LIN {X 0,Y 575.215,Z 1088.939,A -85,B 0,C 180,E1 20584.216,E2 20584.216} C_VEL
LIN {X 0,Y 578.053,Z 1069.285,A -85,B 0,C 180,E1 20581.709,E2 20581.709} C_VEL
LIN {X 0,Y 580.453,Z 1053.893,A -85,B 0,C 180,E1 20579.973,E2 20579.973} C_VEL
LIN {X 0,Y 583.494,Z 1035.186,A -85,B 0,C 180,E1 20578.086,E2 20578.086} C_VEL
LIN {X 0,Y 586.743,Z 1014.887,A -85,B 0,C 180,E1 20576.311,E2 20576.311} C_VEL
LIN {X 0,Y 589.518,Z 997.438,A -85,B 0,C 180,E1 20574.962,E2 20574.962} C_VEL
LIN {X 0,Y 592.71,Z 977.137,A -85,B 0,C 180,E1 20573.573,E2 20573.573} C_VEL
LIN {X 0,Y 595.995,Z 954.418,A -85,B 0,C 180,E1 20572.241,E2 20572.241} C_VEL
LIN {X 0,Y 598.554,Z 935.209,A -85,B 0,C 180,E1 20571.273,E2 20571.273} C_VEL
LIN {X 0,Y 600.798,Z 916.678,A -85,B 0,C 180,E1 20570.463,E2 20570.463} C_VEL
LIN {X 0,Y 603.05,Z 895.538,A -85,B 0,C 180,E1 20569.681,E2 20569.681} C_VEL
LIN {X 0,Y 605.325,Z 869.865,A -85,B 0,C 180,E1 20568.921,E2 20568.921} C_VEL
LIN {X 0,Y 606.783,Z 848.524,A -85,B 0,C 180,E1 20568.434,E2 20568.434} C_VEL
LIN {X 0,Y 607.837,Z 827.107,A -85,B 0,C 180,E1 20568.062,E2 20568.062} C_VEL
LIN {X 0,Y 613.605,Z 599.561,A -85,B 0,C 180,E1 20564.976,E2 20564.976} C_VEL
LIN {X 0,Y 617.781,Z 441.673,A -85,B 0,C 180,E1 20562.787,E2 20562.787} C_VEL
LIN {X 0,Y 611.446,Z 410.233,A -85,B 0,C 180,E1 20561.538,E2 20561.538} C_VEL
LIN {X 0,Y 597.897,Z 389.86,A -85,B 0,C 180,E1 20559.519,E2 20559.519} C_VEL
LIN {X 0,Y 590.526,Z 374.156,A -85,B 0,C 180,E1 20557.07,E2 20557.07} C_VEL
LIN {X 0,Y 583.564,Z 360.458,A -85,B 0,C 180,E1 20554.671,E2 20554.671} C_VEL
LIN {X 0,Y 579.173,Z 351.956,A -85,B 0,C 180,E1 20553.062,E2 20553.062} C_VEL
LIN {X 0,Y 576.456,Z 347.036,A -85,B 0,C 180,E1 20552.058,E2 20552.058} C_VEL
LIN {X 0,Y 574.452,Z 343.015,A -85,B 0,C 180,E1 20551.245,E2 20551.245} C_VEL
LIN {X 0,Y 572.351,Z 339.399,A -85,B 0,C 180,E1 20550.44,E2 20550.44} C_VEL
LIN {X 0,Y 571.332,Z 337.612,A -85,B 0,C 180,E1 20550.035,E2 20550.035} C_VEL
LIN {X 0,Y 569.492,Z 333.982,A -85,B 0,C 180,E1 20549.216,E2 20549.216} C_VEL
LIN {X 0,Y 569.352,Z 333.336,A -85,B 0,C 180,E1 20548.879,E2 20548.879} C_VEL
LIN {X 0,Y 569.379,Z 333.282,A -85,B 0,C 180,E1 20545.595,E2 20545.595} C_VEL
LIN {X 0,Y 569.349,Z 333.278,A -85,B 0,C 180,E1 20542.293,E2 20542.293} C_VEL
LIN {X 0,Y 569.372,Z 333.252,A -85,B 0,C 180,E1 20539.065,E2 20539.065} C_VEL
LIN {X 0,Y 569.379,Z 333.308,A -85,B 0,C 180,E1 20535.691,E2 20535.691} C_VEL
LIN {X 0,Y 569.354,Z 333.245,A -85,B 0,C 180,E1 20532.372,E2 20532.372} C_VEL
LIN {X 0,Y 569.369,Z 333.302,A -85,B 0,C 180,E1 20529.094,E2 20529.094} C_VEL
LIN {X 0,Y 569.369,Z 333.245,A -85,B 0,C 180,E1 20525.745,E2 20525.745} C_VEL
LIN {X 0,Y 569.374,Z 333.291,A -85,B 0,C 180,E1 20522.416,E2 20522.416} C_VEL
LIN {X 0,Y 569.352,Z 333.257,A -85,B 0,C 180,E1 20519.094,E2 20519.094} C_VEL
LIN {X 0,Y 569.373,Z 333.284,A -85,B 0,C 180,E1 20515.871,E2 20515.871} C_VEL
LIN {X 0,Y 569.359,Z 333.264,A -85,B 0,C 180,E1 20512.533,E2 20512.533} C_VEL
LIN {X 0,Y 569.349,Z 333.267,A -85,B 0,C 180,E1 20509.169,E2 20509.169} C_VEL
LIN {X 0,Y 569.382,Z 333.284,A -85,B 0,C 180,E1 20505.871,E2 20505.871} C_VEL
LIN {X 0,Y 569.332,Z 333.255,A -85,B 0,C 180,E1 20502.629,E2 20502.629} C_VEL
LIN {X 0,Y 569.371,Z 333.311,A -85,B 0,C 180,E1 20499.33,E2 20499.33} C_VEL
LIN {X 0,Y 569.337,Z 333.257,A -85,B 0,C 180,E1 20496.175,E2 20496.175} C_VEL
LIN {X 0,Y 569.327,Z 333.282,A -85,B 0,C 180,E1 20492.83,E2 20492.83} C_VEL
LIN {X 0,Y 569.39,Z 333.734,A -85,B 0,C 180,E1 20492.411,E2 20492.411} C_VEL
LIN {X 0,Y 570.987,Z 337.158,A -85,B 0,C 180,E1 20491.669,E2 20491.669} C_VEL
LIN {X 0,Y 572.36,Z 339.239,A -85,B 0,C 180,E1 20491.173,E2 20491.173} C_VEL
LIN {X 0,Y 574.43,Z 343,A -85,B 0,C 180,E1 20490.373,E2 20490.373} C_VEL
LIN {X 0,Y 577.912,Z 349.337,A -85,B 0,C 180,E1 20489.078,E2 20489.078} C_VEL
LIN {X 0,Y 582.608,Z 357.641,A -85,B 0,C 180,E1 20487.508,E2 20487.508} C_VEL
LIN {X 0,Y 592.791,Z 370.97,A -85,B 0,C 180,E1 20485.827,E2 20485.827} C_VEL
LIN {X 0,Y 602.215,Z 383.402,A -85,B 0,C 180,E1 20484.382,E2 20484.382} C_VEL
LIN {X 0,Y 615.574,Z 402.306,A -85,B 0,C 180,E1 20482.459,E2 20482.459} C_VEL
LIN {X 0,Y 622.733,Z 413.094,A -85,B 0,C 180,E1 20481.481,E2 20481.481} C_VEL
LIN {X 0,Y 616.942,Z 613.718,A -85,B 0,C 180,E1 20478.606,E2 20478.606} C_VEL
LIN {X 0,Y 611.425,Z 825.012,A -85,B 0,C 180,E1 20475.663,E2 20475.663} C_VEL
LIN {X 0,Y 610.25,Z 847.871,A -85,B 0,C 180,E1 20475.265,E2 20475.265} C_VEL
LIN {X 0,Y 608.433,Z 874.998,A -85,B 0,C 180,E1 20474.636,E2 20474.636} C_VEL
LIN {X 0,Y 606.238,Z 899.951,A -85,B 0,C 180,E1 20473.882,E2 20473.882} C_VEL
LIN {X 0,Y 604.145,Z 921.03,A -85,B 0,C 180,E1 20473.12,E2 20473.12} C_VEL
LIN {X 0,Y 601.971,Z 941.046,A -85,B 0,C 180,E1 20472.276,E2 20472.276} C_VEL
LIN {X 0,Y 599.598,Z 960.799,A -85,B 0,C 180,E1 20471.327,E2 20471.327} C_VEL
LIN {X 0,Y 596.742,Z 983.005,A -85,B 0,C 180,E1 20470.109,E2 20470.109} C_VEL
LIN {X 0,Y 593.087,Z 1007.09,A -85,B 0,C 180,E1 20468.531,E2 20468.531} C_VEL
LIN {X 0,Y 590.071,Z 1026.218,A -85,B 0,C 180,E1 20467.102,E2 20467.102} C_VEL
LIN {X 0,Y 587.305,Z 1043.431,A -85,B 0,C 180,E1 20465.669,E2 20465.669} C_VEL
LIN {X 0,Y 584.512,Z 1060.71,A -85,B 0,C 180,E1 20464.071,E2 20464.071} C_VEL
LIN {X 0,Y 581.227,Z 1081.272,A -85,B 0,C 180,E1 20461.937,E2 20461.937} C_VEL
LIN {X 0,Y 578.488,Z 1098.828,A -85,B 0,C 180,E1 20459.854,E2 20459.854} C_VEL
LIN {X 0,Y 576.301,Z 1113.378,A -85,B 0,C 180,E1 20457.933,E2 20457.933} C_VEL
LIN {X 0,Y 574.059,Z 1129.58,A -85,B 0,C 180,E1 20455.544,E2 20455.544} C_VEL
LIN {X 0,Y 572.164,Z 1144.275,A -85,B 0,C 180,E1 20453.044,E2 20453.044} C_VEL
LIN {X 0,Y 570.861,Z 1155.779,A -85,B 0,C 180,E1 20450.827,E2 20450.827} C_VEL
LIN {X 0,Y 569.844,Z 1166.361,A -85,B 0,C 180,E1 20448.517,E2 20448.517} C_VEL
LIN {X 0,Y 568.941,Z 1177.381,A -85,B 0,C 180,E1 20445.702,E2 20445.702} C_VEL
LIN {X 0,Y 568.479,Z 1185.17,A -85,B 0,C 180,E1 20443.321,E2 20443.321} C_VEL
LIN {X 0,Y 568.159,Z 1191.597,A -85,B 0,C 180,E1 20440.956,E2 20440.956} C_VEL
LIN {X 0,Y 568.007,Z 1197.191,A -85,B 0,C 180,E1 20438.381,E2 20438.381} C_VEL
LIN {X 0,Y 567.933,Z 1201.538,A -85,B 0,C 180,E1 20435.556,E2 20435.556} C_VEL
LIN {X 0,Y 567.917,Z 1203.848,A -85,B 0,C 180,E1 20433.128,E2 20433.128} C_VEL
LIN {X 0,Y 567.906,Z 1204.804,A -85,B 0,C 180,E1 20430.908,E2 20430.908} C_VEL
LIN {X 0,Y 567.916,Z 1204.736,A -85,B 0,C 180,E1 20428.789,E2 20428.789} C_VEL
LIN {X 0,Y 567.912,Z 1203.507,A -85,B 0,C 180,E1 20426.366,E2 20426.366} C_VEL
LIN {X 0,Y 567.948,Z 1200.335,A -85,B 0,C 180,E1 20423.53,E2 20423.53} C_VEL
LIN {X 0,Y 568.029,Z 1196.126,A -85,B 0,C 180,E1 20421.089,E2 20421.089} C_VEL
LIN {X 0,Y 568.191,Z 1190.833,A -85,B 0,C 180,E1 20418.736,E2 20418.736} C_VEL
LIN {X 0,Y 568.577,Z 1183.47,A -85,B 0,C 180,E1 20416.106,E2 20416.106} C_VEL
LIN {X 0,Y 569.205,Z 1173.918,A -85,B 0,C 180,E1 20413.361,E2 20413.361} C_VEL
LIN {X 0,Y 570.006,Z 1164.527,A -85,B 0,C 180,E1 20411.063,E2 20411.063} C_VEL
LIN {X 0,Y 571.044,Z 1154.238,A -85,B 0,C 180,E1 20408.857,E2 20408.857} C_VEL
LIN {X 0,Y 572.692,Z 1140.174,A -85,B 0,C 180,E1 20406.215,E2 20406.215} C_VEL
LIN {X 0,Y 574.534,Z 1125.776,A -85,B 0,C 180,E1 20403.877,E2 20403.877} C_VEL
LIN {X 0,Y 576.538,Z 1111.833,A -85,B 0,C 180,E1 20401.854,E2 20401.854} C_VEL
LIN {X 0,Y 579.024,Z 1095.329,A -85,B 0,C 180,E1 20399.704,E2 20399.704} C_VEL
LIN {X 0,Y 582.167,Z 1075.37,A -85,B 0,C 180,E1 20397.428,E2 20397.428} C_VEL
LIN {X 0,Y 584.784,Z 1059.04,A -85,B 0,C 180,E1 20395.769,E2 20395.769} C_VEL
LIN {X 0,Y 587.477,Z 1042.38,A -85,B 0,C 180,E1 20394.24,E2 20394.24} C_VEL
LIN {X 0,Y 590.375,Z 1024.362,A -85,B 0,C 180,E1 20392.752,E2 20392.752} C_VEL
LIN {X 0,Y 594.049,Z 1001.028,A -85,B 0,C 180,E1 20391.044,E2 20391.044} C_VEL
LIN {X 0,Y 597.088,Z 980.227,A -85,B 0,C 180,E1 20389.73,E2 20389.73} C_VEL
LIN {X 0,Y 599.74,Z 959.604,A -85,B 0,C 180,E1 20388.612,E2 20388.612} C_VEL
LIN {X 0,Y 602.123,Z 939.747,A -85,B 0,C 180,E1 20387.666,E2 20387.666} C_VEL
LIN {X 0,Y 604.431,Z 918.348,A -85,B 0,C 180,E1 20386.775,E2 20386.775} C_VEL
LIN {X 0,Y 607.062,Z 891.208,A -85,B 0,C 180,E1 20385.832,E2 20385.832} C_VEL
LIN {X 0,Y 609.036,Z 866.174,A -85,B 0,C 180,E1 20385.144,E2 20385.144} C_VEL
LIN {X 0,Y 610.419,Z 844.794,A -85,B 0,C 180,E1 20384.674,E2 20384.674} C_VEL
LIN {X 0,Y 611.52,Z 822.48,A -85,B 0,C 180,E1 20384.299,E2 20384.299} C_VEL
LIN {X 0,Y 617.232,Z 602.035,A -85,B 0,C 180,E1 20381.232,E2 20381.232} C_VEL
LIN {X 0,Y 622.721,Z 412.863,A -85,B 0,C 180,E1 20378.514,E2 20378.514} C_VEL
LIN {X 0,Y 607.623,Z 390.884,A -85,B 0,C 180,E1 20376.416,E2 20376.416} C_VEL
LIN {X 0,Y 594.34,Z 372.937,A -85,B 0,C 180,E1 20374.421,E2 20374.421} C_VEL
LIN {X 0,Y 586.055,Z 362.24,A -85,B 0,C 180,E1 20373.091,E2 20373.091} C_VEL
LIN {X 0,Y 582.119,Z 357.051,A -85,B 0,C 180,E1 20372.406,E2 20372.406} C_VEL
LIN {X 0,Y 579.52,Z 352.35,A -85,B 0,C 180,E1 20371.52,E2 20371.52} C_VEL
LIN {X 0,Y 576.62,Z 347.132,A -85,B 0,C 180,E1 20370.479,E2 20370.479} C_VEL
LIN {X 0,Y 574.387,Z 342.955,A -85,B 0,C 180,E1 20369.629,E2 20369.629} C_VEL
LIN {X 0,Y 572.332,Z 339.159,A -85,B 0,C 180,E1 20368.828,E2 20368.828} C_VEL
LIN {X 0,Y 569.532,Z 334.345,A -85,B 0,C 180,E1 20367.726,E2 20367.726} C_VEL
LIN {X 0,Y 569.344,Z 333.479,A -85,B 0,C 180,E1 20367.509,E2 20367.509} C_VEL
LIN {X 0,Y 569.38,Z 333.261,A -85,B 0,C 180,E1 20364.374,E2 20364.374} C_VEL
LIN {X 0,Y 569.331,Z 333.303,A -85,B 0,C 180,E1 20361.162,E2 20361.162} C_VEL
LIN {X 0,Y 569.357,Z 333.249,A -85,B 0,C 180,E1 20357.855,E2 20357.855} C_VEL
LIN {X 0,Y 569.367,Z 333.303,A -85,B 0,C 180,E1 20354.619,E2 20354.619} C_VEL
LIN {X 0,Y 569.339,Z 333.255,A -85,B 0,C 180,E1 20351.344,E2 20351.344} C_VEL
LIN {X 0,Y 569.377,Z 333.289,A -85,B 0,C 180,E1 20348.178,E2 20348.178} C_VEL
LIN {X 0,Y 569.344,Z 333.261,A -85,B 0,C 180,E1 20344.937,E2 20344.937} C_VEL
LIN {X 0,Y 569.376,Z 333.281,A -85,B 0,C 180,E1 20341.711,E2 20341.711} C_VEL
LIN {X 0,Y 569.368,Z 333.263,A -85,B 0,C 180,E1 20338.39,E2 20338.39} C_VEL
LIN {X 0,Y 569.359,Z 333.267,A -85,B 0,C 180,E1 20335.063,E2 20335.063} C_VEL
LIN {X 0,Y 569.364,Z 333.27,A -85,B 0,C 180,E1 20331.822,E2 20331.822} C_VEL
LIN {X 0,Y 569.363,Z 333.256,A -85,B 0,C 180,E1 20328.554,E2 20328.554} C_VEL
LIN {X 0,Y 569.381,Z 333.294,A -85,B 0,C 180,E1 20325.144,E2 20325.144} C_VEL
LIN {X 0,Y 569.357,Z 333.249,A -85,B 0,C 180,E1 20321.784,E2 20321.784} C_VEL
LIN {X 0,Y 569.375,Z 333.305,A -85,B 0,C 180,E1 20318.467,E2 20318.467} C_VEL
LIN {X 0,Y 569.35,Z 333.261,A -85,B 0,C 180,E1 20315.182,E2 20315.182} C_VEL
LIN {X 0,Y 569.362,Z 333.258,A -85,B 0,C 180,E1 20311.834,E2 20311.834} C_VEL
LIN {X 0,Y 569.43,Z 333.642,A -85,B 0,C 180,E1 20310.739,E2 20310.739} C_VEL
LIN {X 0,Y 571.05,Z 337.255,A -85,B 0,C 180,E1 20309.948,E2 20309.948} C_VEL
LIN {X 0,Y 572.364,Z 339.417,A -85,B 0,C 180,E1 20309.445,E2 20309.445} C_VEL
LIN {X 0,Y 574.475,Z 343.031,A -85,B 0,C 180,E1 20308.64,E2 20308.64} C_VEL
LIN {X 0,Y 577.257,Z 348.085,A -85,B 0,C 180,E1 20307.581,E2 20307.581} C_VEL
LIN {X 0,Y 584.777,Z 362.651,A -85,B 0,C 180,E1 20304.814,E2 20304.814} C_VEL
LIN {X 0,Y 591.129,Z 375.567,A -85,B 0,C 180,E1 20302.609,E2 20302.609} C_VEL
LIN {X 0,Y 598.317,Z 390.561,A -85,B 0,C 180,E1 20300.297,E2 20300.297} C_VEL
LIN {X 0,Y 611.582,Z 410.455,A -85,B 0,C 180,E1 20298.348,E2 20298.348} C_VEL
LIN {X 0,Y 617.828,Z 442.453,A -85,B 0,C 180,E1 20297.101,E2 20297.101} C_VEL
LIN {X 0,Y 612.398,Z 646.343,A -85,B 0,C 180,E1 20294.298,E2 20294.298} C_VEL
LIN {X 0,Y 611.526,Z 654.049,A -85,B 0,C 180,E1 20294.26,E2 20294.26} C_VEL
LIN {X 0,Y 606.683,Z 674.681,A -85,B 0,C 180,E1 20294.41,E2 20294.41} C_VEL
LIN {X 0,Y 605.99,Z 681.294,A -85,B 0,C 180,E1 20294.372,E2 20294.372} C_VEL
LIN {X 0,Y 601.978,Z 831.027,A -85,B 0,C 180,E1 20292.324,E2 20292.324} C_VEL
LIN {X 0,Y 600.473,Z 857.229,A -85,B 0,C 180,E1 20291.836,E2 20291.836} C_VEL
LIN {X 0,Y 598.478,Z 881.561,A -85,B 0,C 180,E1 20291.203,E2 20291.203} C_VEL
LIN {X 0,Y 596.403,Z 902.748,A -85,B 0,C 180,E1 20290.515,E2 20290.515} C_VEL
LIN {X 0,Y 593.623,Z 927.269,A -85,B 0,C 180,E1 20289.546,E2 20289.546} C_VEL
LIN {X 0,Y 590.628,Z 949.512,A -85,B 0,C 180,E1 20288.473,E2 20288.473} C_VEL
LIN {X 0,Y 587.921,Z 967.877,A -85,B 0,C 180,E1 20287.445,E2 20287.445} C_VEL
LIN {X 0,Y 584.637,Z 988.821,A -85,B 0,C 180,E1 20286.099,E2 20286.099} C_VEL
LIN {X 0,Y 580.995,Z 1010.481,A -85,B 0,C 180,E1 20284.476,E2 20284.476} C_VEL
LIN {X 0,Y 578.043,Z 1027.611,A -85,B 0,C 180,E1 20283.016,E2 20283.016} C_VEL
LIN {X 0,Y 575.112,Z 1044.691,A -85,B 0,C 180,E1 20281.388,E2 20281.388} C_VEL
LIN {X 0,Y 571.696,Z 1064.709,A -85,B 0,C 180,E1 20279.207,E2 20279.207} C_VEL
LIN {X 0,Y 569.31,Z 1079.368,A -85,B 0,C 180,E1 20277.397,E2 20277.397} C_VEL
LIN {X 0,Y 567.05,Z 1094.053,A -85,B 0,C 180,E1 20275.371,E2 20275.371} C_VEL
LIN {X 0,Y 564.814,Z 1110.511,A -85,B 0,C 180,E1 20272.811,E2 20272.811} C_VEL
LIN {X 0,Y 563.394,Z 1122.352,A -85,B 0,C 180,E1 20270.722,E2 20270.722} C_VEL
LIN {X 0,Y 562.109,Z 1134.782,A -85,B 0,C 180,E1 20268.214,E2 20268.214} C_VEL
LIN {X 0,Y 561.215,Z 1144.797,A -85,B 0,C 180,E1 20265.819,E2 20265.819} C_VEL
LIN {X 0,Y 560.651,Z 1152.781,A -85,B 0,C 180,E1 20263.595,E2 20263.595} C_VEL
LIN {X 0,Y 560.226,Z 1160.757,A -85,B 0,C 180,E1 20260.906,E2 20260.906} C_VEL
LIN {X 0,Y 560.04,Z 1166.03,A -85,B 0,C 180,E1 20258.625,E2 20258.625} C_VEL
LIN {X 0,Y 559.956,Z 1169.917,A -85,B 0,C 180,E1 20256.459,E2 20256.459} C_VEL
LIN {X 0,Y 559.914,Z 1172.807,A -85,B 0,C 180,E1 20254.199,E2 20254.199} C_VEL
LIN {X 0,Y 559.902,Z 1174.653,A -85,B 0,C 180,E1 20251.535,E2 20251.535} C_VEL
LIN {X 0,Y 559.897,Z 1174.856,A -85,B 0,C 180,E1 20249.284,E2 20249.284} C_VEL
LIN {X 0,Y 559.906,Z 1173.968,A -85,B 0,C 180,E1 20247.134,E2 20247.134} C_VEL
LIN {X 0,Y 559.916,Z 1171.999,A -85,B 0,C 180,E1 20244.98,E2 20244.98} C_VEL
LIN {X 0,Y 559.979,Z 1168.276,A -85,B 0,C 180,E1 20242.407,E2 20242.407} C_VEL
LIN {X 0,Y 560.122,Z 1163.013,A -85,B 0,C 180,E1 20239.925,E2 20239.925} C_VEL
LIN {X 0,Y 560.401,Z 1157.204,A -85,B 0,C 180,E1 20237.742,E2 20237.742} C_VEL
LIN {X 0,Y 560.842,Z 1149.832,A -85,B 0,C 180,E1 20235.441,E2 20235.441} C_VEL
LIN {X 0,Y 561.64,Z 1139.632,A -85,B 0,C 180,E1 20232.811,E2 20232.811} C_VEL
LIN {X 0,Y 562.562,Z 1130.009,A -85,B 0,C 180,E1 20230.696,E2 20230.696} C_VEL
LIN {X 0,Y 563.78,Z 1119.028,A -85,B 0,C 180,E1 20228.571,E2 20228.571} C_VEL
LIN {X 0,Y 565.678,Z 1103.775,A -85,B 0,C 180,E1 20226.012,E2 20226.012} C_VEL
LIN {X 0,Y 568.094,Z 1087.181,A -85,B 0,C 180,E1 20223.558,E2 20223.558} C_VEL
LIN {X 0,Y 570.85,Z 1069.89,A -85,B 0,C 180,E1 20221.32,E2 20221.32} C_VEL
LIN {X 0,Y 573.487,Z 1054.105,A -85,B 0,C 180,E1 20219.512,E2 20219.512} C_VEL
LIN {X 0,Y 576.522,Z 1036.52,A -85,B 0,C 180,E1 20217.713,E2 20217.713} C_VEL
LIN {X 0,Y 580.176,Z 1015.196,A -85,B 0,C 180,E1 20215.818,E2 20215.818} C_VEL
LIN {X 0,Y 583.119,Z 997.822,A -85,B 0,C 180,E1 20214.459,E2 20214.459} C_VEL
LIN {X 0,Y 586.335,Z 978.32,A -85,B 0,C 180,E1 20213.111,E2 20213.111} C_VEL
LIN {X 0,Y 589.918,Z 954.728,A -85,B 0,C 180,E1 20211.714,E2 20211.714} C_VEL
LIN {X 0,Y 592.557,Z 935.478,A -85,B 0,C 180,E1 20210.745,E2 20210.745} C_VEL
LIN {X 0,Y 594.882,Z 916.705,A -85,B 0,C 180,E1 20209.929,E2 20209.929} C_VEL
LIN {X 0,Y 597.121,Z 896.268,A -85,B 0,C 180,E1 20209.171,E2 20209.171} C_VEL
LIN {X 0,Y 599.501,Z 870.507,A -85,B 0,C 180,E1 20208.402,E2 20208.402} C_VEL
LIN {X 0,Y 601.046,Z 848.667,A -85,B 0,C 180,E1 20207.901,E2 20207.901} C_VEL
LIN {X 0,Y 602.135,Z 827.355,A -85,B 0,C 180,E1 20207.53,E2 20207.53} C_VEL
LIN {X 0,Y 608.258,Z 596.705,A -85,B 0,C 180,E1 20204.381,E2 20204.381} C_VEL
LIN {X 0,Y 612.512,Z 443.576,A -85,B 0,C 180,E1 20202.242,E2 20202.242} C_VEL
LIN {X 0,Y 606.894,Z 415.194,A -85,B 0,C 180,E1 20201.1,E2 20201.1} C_VEL
LIN {X 0,Y 593.37,Z 395.038,A -85,B 0,C 180,E1 20199.067,E2 20199.067} C_VEL
LIN {X 0,Y 589.348,Z 388.963,A -85,B 0,C 180,E1 20198.386,E2 20198.386} C_VEL
LIN {X 0,Y 582.296,Z 374.276,A -85,B 0,C 180,E1 20195.963,E2 20195.963} C_VEL
LIN {X 0,Y 576.415,Z 362.589,A -85,B 0,C 180,E1 20193.837,E2 20193.837} C_VEL
LIN {X 0,Y 571.585,Z 353.4,A -85,B 0,C 180,E1 20192.009,E2 20192.009} C_VEL
LIN {X 0,Y 568.98,Z 348.618,A -85,B 0,C 180,E1 20190.991,E2 20190.991} C_VEL
LIN {X 0,Y 566.206,Z 343.58,A -85,B 0,C 180,E1 20189.868,E2 20189.868} C_VEL
LIN {X 0,Y 563.74,Z 339.019,A -85,B 0,C 180,E1 20188.815,E2 20188.815} C_VEL
LIN {X 0,Y 561.82,Z 335.92,A -85,B 0,C 180,E1 20188.025,E2 20188.025} C_VEL
LIN {X 0,Y 561.468,Z 334.458,A -85,B 0,C 180,E1 20187.656,E2 20187.656} C_VEL
LIN {X 0,Y 561.403,Z 334.243,A -85,B 0,C 180,E1 20184.406,E2 20184.406} C_VEL
LIN {X 0,Y 561.441,Z 334.297,A -85,B 0,C 180,E1 20181.062,E2 20181.062} C_VEL
LIN {X 0,Y 561.433,Z 334.239,A -85,B 0,C 180,E1 20177.674,E2 20177.674} C_VEL
LIN {X 0,Y 561.417,Z 334.27,A -85,B 0,C 180,E1 20174.439,E2 20174.439} C_VEL
LIN {X 0,Y 561.427,Z 334.251,A -85,B 0,C 180,E1 20171.097,E2 20171.097} C_VEL
LIN {X 0,Y 561.434,Z 334.245,A -85,B 0,C 180,E1 20167.779,E2 20167.779} C_VEL
LIN {X 0,Y 561.431,Z 334.271,A -85,B 0,C 180,E1 20164.392,E2 20164.392} C_VEL
LIN {X 0,Y 561.414,Z 334.24,A -85,B 0,C 180,E1 20161.123,E2 20161.123} C_VEL
LIN {X 0,Y 561.434,Z 334.284,A -85,B 0,C 180,E1 20157.857,E2 20157.857} C_VEL
LIN {X 0,Y 561.419,Z 334.236,A -85,B 0,C 180,E1 20154.584,E2 20154.584} C_VEL
LIN {X 0,Y 561.416,Z 334.294,A -85,B 0,C 180,E1 20151.189,E2 20151.189} C_VEL
LIN {X 0,Y 561.434,Z 334.23,A -85,B 0,C 180,E1 20147.869,E2 20147.869} C_VEL
LIN {X 0,Y 561.403,Z 334.299,A -85,B 0,C 180,E1 20144.611,E2 20144.611} C_VEL
LIN {X 0,Y 561.419,Z 334.241,A -85,B 0,C 180,E1 20141.302,E2 20141.302} C_VEL
LIN {X 0,Y 561.409,Z 334.262,A -85,B 0,C 180,E1 20138.146,E2 20138.146} C_VEL
LIN {X 0,Y 561.39,Z 334.28,A -85,B 0,C 180,E1 20134.794,E2 20134.794} C_VEL
LIN {X 0,Y 561.488,Z 334.675,A -85,B 0,C 180,E1 20133.815,E2 20133.815} C_VEL
LIN {X 0,Y 563.184,Z 338.387,A -85,B 0,C 180,E1 20132.967,E2 20132.967} C_VEL
LIN {X 0,Y 564.507,Z 340.35,A -85,B 0,C 180,E1 20132.464,E2 20132.464} C_VEL
LIN {X 0,Y 566.511,Z 343.879,A -85,B 0,C 180,E1 20131.655,E2 20131.655} C_VEL
LIN {X 0,Y 567.71,Z 346.299,A -85,B 0,C 180,E1 20131.145,E2 20131.145} C_VEL
LIN {X 0,Y 570.374,Z 350.886,A -85,B 0,C 180,E1 20130.141,E2 20130.141} C_VEL
LIN {X 0,Y 573.266,Z 356.395,A -85,B 0,C 180,E1 20129.033,E2 20129.033} C_VEL
LIN {X 0,Y 575.118,Z 359.033,A -85,B 0,C 180,E1 20128.562,E2 20128.562} C_VEL
LIN {X 0,Y 585.729,Z 372.597,A -85,B 0,C 180,E1 20126.742,E2 20126.742} C_VEL
LIN {X 0,Y 596.398,Z 386.71,A -85,B 0,C 180,E1 20125.043,E2 20125.043} C_VEL
LIN {X 0,Y 608.942,Z 404.374,A -85,B 0,C 180,E1 20123.178,E2 20123.178} C_VEL
LIN {X 0,Y 617.393,Z 417.147,A -85,B 0,C 180,E1 20121.988,E2 20121.988} C_VEL
LIN {X 0,Y 611.149,Z 620.112,A -85,B 0,C 180,E1 20119.051,E2 20119.051} C_VEL
LIN {X 0,Y 605.333,Z 827.696,A -85,B 0,C 180,E1 20116.126,E2 20116.126} C_VEL
LIN {X 0,Y 603.724,Z 855.846,A -85,B 0,C 180,E1 20115.601,E2 20115.601} C_VEL
LIN {X 0,Y 601.702,Z 881.502,A -85,B 0,C 180,E1 20114.947,E2 20114.947} C_VEL
LIN {X 0,Y 599.75,Z 902.878,A -85,B 0,C 180,E1 20114.276,E2 20114.276} C_VEL
LIN {X 0,Y 597.6,Z 923.472,A -85,B 0,C 180,E1 20113.511,E2 20113.511} C_VEL
LIN {X 0,Y 594.924,Z 946.696,A -85,B 0,C 180,E1 20112.503,E2 20112.503} C_VEL
LIN {X 0,Y 591.532,Z 972.526,A -85,B 0,C 180,E1 20111.176,E2 20111.176} C_VEL
LIN {X 0,Y 588.613,Z 993.178,A -85,B 0,C 180,E1 20109.949,E2 20109.949} C_VEL
LIN {X 0,Y 586.118,Z 1010.033,A -85,B 0,C 180,E1 20108.824,E2 20108.824} C_VEL
LIN {X 0,Y 583.224,Z 1027.551,A -85,B 0,C 180,E1 20107.489,E2 20107.489} C_VEL
LIN {X 0,Y 580.229,Z 1045.255,A -85,B 0,C 180,E1 20105.988,E2 20105.988} C_VEL
LIN {X 0,Y 576.748,Z 1065.847,A -85,B 0,C 180,E1 20104.035,E2 20104.035} C_VEL
LIN {X 0,Y 573.492,Z 1084.881,A -85,B 0,C 180,E1 20101.96,E2 20101.96} C_VEL
LIN {X 0,Y 570.938,Z 1100.517,A -85,B 0,C 180,E1 20100.057,E2 20100.057} C_VEL
LIN {X 0,Y 568.539,Z 1115.687,A -85,B 0,C 180,E1 20098.006,E2 20098.006} C_VEL
LIN {X 0,Y 565.982,Z 1133.186,A -85,B 0,C 180,E1 20095.31,E2 20095.31} C_VEL
LIN {X 0,Y 564.313,Z 1145.583,A -85,B 0,C 180,E1 20093.131,E2 20093.131} C_VEL
LIN {X 0,Y 562.963,Z 1156.91,A -85,B 0,C 180,E1 20090.894,E2 20090.894} C_VEL
LIN {X 0,Y 561.754,Z 1169.038,A -85,B 0,C 180,E1 20088.149,E2 20088.149} C_VEL
LIN {X 0,Y 560.945,Z 1178.45,A -85,B 0,C 180,E1 20085.614,E2 20085.614} C_VEL
LIN {X 0,Y 560.49,Z 1185.773,A -85,B 0,C 180,E1 20083.304,E2 20083.304} C_VEL
LIN {X 0,Y 560.158,Z 1192.357,A -85,B 0,C 180,E1 20080.802,E2 20080.802} C_VEL
LIN {X 0,Y 559.997,Z 1198.08,A -85,B 0,C 180,E1 20078.005,E2 20078.005} C_VEL
LIN {X 0,Y 559.93,Z 1201.763,A -85,B 0,C 180,E1 20075.431,E2 20075.431} C_VEL
LIN {X 0,Y 559.916,Z 1203.913,A -85,B 0,C 180,E1 20073.071,E2 20073.071} C_VEL
LIN {X 0,Y 559.902,Z 1204.827,A -85,B 0,C 180,E1 20070.818,E2 20070.818} C_VEL
LIN {X 0,Y 559.912,Z 1204.69,A -85,B 0,C 180,E1 20068.567,E2 20068.567} C_VEL
LIN {X 0,Y 559.917,Z 1203.193,A -85,B 0,C 180,E1 20065.904,E2 20065.904} C_VEL
LIN {X 0,Y 559.951,Z 1200.013,A -85,B 0,C 180,E1 20063.232,E2 20063.232} C_VEL
LIN {X 0,Y 560.042,Z 1195.916,A -85,B 0,C 180,E1 20060.857,E2 20060.857} C_VEL
LIN {X 0,Y 560.237,Z 1190.575,A -85,B 0,C 180,E1 20058.469,E2 20058.469} C_VEL
LIN {X 0,Y 560.658,Z 1183.006,A -85,B 0,C 180,E1 20055.752,E2 20055.752} C_VEL
LIN {X 0,Y 561.334,Z 1173.512,A -85,B 0,C 180,E1 20053.015,E2 20053.015} C_VEL
LIN {X 0,Y 562.169,Z 1164.526,A -85,B 0,C 180,E1 20050.789,E2 20050.789} C_VEL
LIN {X 0,Y 563.288,Z 1154.236,A -85,B 0,C 180,E1 20048.551,E2 20048.551} C_VEL
LIN {X 0,Y 565.044,Z 1140.172,A -85,B 0,C 180,E1 20045.872,E2 20045.872} C_VEL
LIN {X 0,Y 567.02,Z 1125.774,A -85,B 0,C 180,E1 20043.504,E2 20043.504} C_VEL
LIN {X 0,Y 569.139,Z 1111.824,A -85,B 0,C 180,E1 20041.453,E2 20041.453} C_VEL
LIN {X 0,Y 571.756,Z 1095.442,A -85,B 0,C 180,E1 20039.293,E2 20039.293} C_VEL
LIN {X 0,Y 575.042,Z 1075.825,A -85,B 0,C 180,E1 20037.027,E2 20037.027} C_VEL
LIN {X 0,Y 577.883,Z 1059.039,A -85,B 0,C 180,E1 20035.302,E2 20035.302} C_VEL
LIN {X 0,Y 580.647,Z 1042.812,A -85,B 0,C 180,E1 20033.797,E2 20033.797} C_VEL
LIN {X 0,Y 583.452,Z 1026.201,A -85,B 0,C 180,E1 20032.404,E2 20032.404} C_VEL
LIN {X 0,Y 586.374,Z 1008.45,A -85,B 0,C 180,E1 20031.064,E2 20031.064} C_VEL
LIN {X 0,Y 589.807,Z 985.49,A -85,B 0,C 180,E1 20029.569,E2 20029.569} C_VEL
LIN {X 0,Y 593.095,Z 960.885,A -85,B 0,C 180,E1 20028.202,E2 20028.202} C_VEL
LIN {X 0,Y 595.621,Z 940.817,A -85,B 0,C 180,E1 20027.231,E2 20027.231} C_VEL
LIN {X 0,Y 597.888,Z 920.795,A -85,B 0,C 180,E1 20026.382,E2 20026.382} C_VEL
LIN {X 0,Y 600.01,Z 900.295,A -85,B 0,C 180,E1 20025.636,E2 20025.636} C_VEL
LIN {X 0,Y 602.301,Z 875.116,A -85,B 0,C 180,E1 20024.872,E2 20024.872} C_VEL
LIN {X 0,Y 604.209,Z 847.803,A -85,B 0,C 180,E1 20024.234,E2 20024.234} C_VEL
LIN {X 0,Y 605.42,Z 825.368,A -85,B 0,C 180,E1 20023.839,E2 20023.839} C_VEL
LIN {X 0,Y 611.611,Z 604.458,A -85,B 0,C 180,E1 20020.725,E2 20020.725} C_VEL
LIN {X 0,Y 617.365,Z 416.812,A -85,B 0,C 180,E1 20018.005,E2 20018.005} C_VEL
LIN {X 0,Y 603.07,Z 395.945,A -85,B 0,C 180,E1 20015.969,E2 20015.969} C_VEL
LIN {X 0,Y 590.852,Z 379.325,A -85,B 0,C 180,E1 20014.095,E2 20014.095} C_VEL
LIN {X 0,Y 582.515,Z 368.515,A -85,B 0,C 180,E1 20012.731,E2 20012.731} C_VEL
LIN {X 0,Y 574.7,Z 358.569,A -85,B 0,C 180,E1 20011.376,E2 20011.376} C_VEL
LIN {X 0,Y 572.523,Z 354.643,A -85,B 0,C 180,E1 20010.662,E2 20010.662} C_VEL
LIN {X 0,Y 569.277,Z 348.936,A -85,B 0,C 180,E1 20009.459,E2 20009.459} C_VEL
LIN {X 0,Y 567.191,Z 344.888,A -85,B 0,C 180,E1 20008.609,E2 20008.609} C_VEL
LIN {X 0,Y 564.669,Z 340.791,A -85,B 0,C 180,E1 20007.642,E2 20007.642} C_VEL
LIN {X 0,Y 563.71,Z 339.007,A -85,B 0,C 180,E1 20007.235,E2 20007.235} C_VEL
LIN {X 0,Y 561.752,Z 335.695,A -85,B 0,C 180,E1 20006.423,E2 20006.423} C_VEL
LIN {X 0,Y 561.442,Z 334.453,A -85,B 0,C 180,E1 20006.097,E2 20006.097} C_VEL
LIN {X 0,Y 561.397,Z 334.242,A -85,B 0,C 180,E1 20002.956,E2 20002.956} C_VEL
LIN {X 0,Y 561.397,Z 334.267,A -85,B 0,C 180,E1 19999.579,E2 19999.579} C_VEL
LIN {X 0,Y 561.44,Z 334.259,A -85,B 0,C 180,E1 19996.343,E2 19996.343} C_VEL
LIN {X 0,Y 561.395,Z 334.247,A -85,B 0,C 180,E1 19993.178,E2 19993.178} C_VEL
LIN {X 0,Y 561.439,Z 334.282,A -85,B 0,C 180,E1 19989.844,E2 19989.844} C_VEL
LIN {X 0,Y 561.421,Z 334.233,A -85,B 0,C 180,E1 19986.545,E2 19986.545} C_VEL
LIN {X 0,Y 561.416,Z 334.297,A -85,B 0,C 180,E1 19983.165,E2 19983.165} C_VEL
LIN {X 0,Y 561.429,Z 334.228,A -85,B 0,C 180,E1 19979.898,E2 19979.898} C_VEL
LIN {X 0,Y 561.428,Z 334.298,A -85,B 0,C 180,E1 19976.528,E2 19976.528} C_VEL
LIN {X 0,Y 561.427,Z 334.227,A -85,B 0,C 180,E1 19973.147,E2 19973.147} C_VEL
LIN {X 0,Y 561.428,Z 334.286,A -85,B 0,C 180,E1 19969.845,E2 19969.845} C_VEL
LIN {X 0,Y 561.425,Z 334.238,A -85,B 0,C 180,E1 19966.508,E2 19966.508} C_VEL
LIN {X 0,Y 561.428,Z 334.264,A -85,B 0,C 180,E1 19963.231,E2 19963.231} C_VEL
LIN {X 0,Y 561.42,Z 334.267,A -85,B 0,C 180,E1 19959.787,E2 19959.787} C_VEL
LIN {X 0,Y 561.434,Z 334.238,A -85,B 0,C 180,E1 19956.518,E2 19956.518} C_VEL
LIN {X 0,Y 561.413,Z 334.288,A -85,B 0,C 180,E1 19953.218,E2 19953.218} C_VEL
LIN {X 0,Y 561.498,Z 334.642,A -85,B 0,C 180,E1 19952.127,E2 19952.127} C_VEL
LIN {X 0,Y 563.037,Z 338.181,A -85,B 0,C 180,E1 19951.316,E2 19951.316} C_VEL
LIN {X 0,Y 564.348,Z 339.883,A -85,B 0,C 180,E1 19950.841,E2 19950.841} C_VEL
LIN {X 0,Y 566.213,Z 343.597,A -85,B 0,C 180,E1 19950.016,E2 19950.016} C_VEL
LIN {X 0,Y 567.237,Z 345.362,A -85,B 0,C 180,E1 19949.608,E2 19949.608} C_VEL
LIN {X 0,Y 569.309,Z 349.008,A -85,B 0,C 180,E1 19948.794,E2 19948.794} C_VEL
LIN {X 0,Y 575.007,Z 359.87,A -85,B 0,C 180,E1 19946.582,E2 19946.582} C_VEL
LIN {X 0,Y 581.514,Z 372.573,A -85,B 0,C 180,E1 19944.224,E2 19944.224} C_VEL
LIN {X 0,Y 589.124,Z 388.427,A -85,B 0,C 180,E1 19941.596,E2 19941.596} C_VEL
LIN {X 0,Y 591.105,Z 391.782,A -85,B 0,C 180,E1 19941.191,E2 19941.191} C_VEL
LIN {X 0,Y 601.739,Z 407.433,A -85,B 0,C 180,E1 19939.558,E2 19939.558} C_VEL
LIN {X 0,Y 607.139,Z 415.899,A -85,B 0,C 180,E1 19938.763,E2 19938.763} C_VEL
LIN {X 0,Y 612.555,Z 444.674,A -85,B 0,C 180,E1 19937.64,E2 19937.64} C_VEL
LIN {X 0,Y 606.02,Z 680.12,A -85,B 0,C 180,E1 19934.388,E2 19934.388} C_VEL
LIN {X 0,Y 605.99,Z 681.294,A -85,B 0,C 180,E1 19934.372,E2 19934.372} C_VEL
LIN {X 0,Y 605.105,Z 688.998,A -85,B 0,C 180,E1 19934.335,E2 19934.335} C_VEL
LIN {X 0,Y 600.263,Z 709.624,A -85,B 0,C 180,E1 19934.487,E2 19934.487} C_VEL
LIN {X 0,Y 599.552,Z 716.236,A -85,B 0,C 180,E1 19934.451,E2 19934.451} C_VEL
LIN {X 0,Y 596.298,Z 831.418,A -85,B 0,C 180,E1 19932.862,E2 19932.862} C_VEL
LIN {X 0,Y 594.679,Z 858.105,A -85,B 0,C 180,E1 19932.358,E2 19932.358} C_VEL
LIN {X 0,Y 592.652,Z 881.922,A -85,B 0,C 180,E1 19931.734,E2 19931.734} C_VEL
LIN {X 0,Y 590.489,Z 903.211,A -85,B 0,C 180,E1 19931.04,E2 19931.04} C_VEL
LIN {X 0,Y 587.513,Z 928.277,A -85,B 0,C 180,E1 19930.039,E2 19930.039} C_VEL
LIN {X 0,Y 584.556,Z 949.559,A -85,B 0,C 180,E1 19929.011,E2 19929.011} C_VEL
LIN {X 0,Y 581.621,Z 968.985,A -85,B 0,C 180,E1 19927.922,E2 19927.922} C_VEL
LIN {X 0,Y 578.105,Z 990.788,A -85,B 0,C 180,E1 19926.511,E2 19926.511} C_VEL
LIN {X 0,Y 574.391,Z 1011.577,A -85,B 0,C 180,E1 19924.924,E2 19924.924} C_VEL
LIN {X 0,Y 571.297,Z 1028.55,A -85,B 0,C 180,E1 19923.457,E2 19923.457} C_VEL
LIN {X 0,Y 567.91,Z 1047.173,A -85,B 0,C 180,E1 19921.646,E2 19921.646} C_VEL
LIN {X 0,Y 564.533,Z 1065.661,A -85,B 0,C 180,E1 19919.581,E2 19919.581} C_VEL
LIN {X 0,Y 561.902,Z 1080.77,A -85,B 0,C 180,E1 19917.674,E2 19917.674} C_VEL
LIN {X 0,Y 559.178,Z 1097.467,A -85,B 0,C 180,E1 19915.3,E2 19915.3} C_VEL
LIN {X 0,Y 557.098,Z 1111.267,A -85,B 0,C 180,E1 19913.033,E2 19913.033} C_VEL
LIN {X 0,Y 555.246,Z 1125.973,A -85,B 0,C 180,E1 19910.338,E2 19910.338} C_VEL
LIN {X 0,Y 554.001,Z 1137.406,A -85,B 0,C 180,E1 19907.868,E2 19907.868} C_VEL
LIN {X 0,Y 553.19,Z 1146.417,A -85,B 0,C 180,E1 19905.624,E2 19905.624} C_VEL
LIN {X 0,Y 552.528,Z 1155.732,A -85,B 0,C 180,E1 19902.861,E2 19902.861} C_VEL
LIN {X 0,Y 552.19,Z 1162.123,A -85,B 0,C 180,E1 19900.5,E2 19900.5} C_VEL
LIN {X 0,Y 552.033,Z 1166.86,A -85,B 0,C 180,E1 19898.332,E2 19898.332} C_VEL
LIN {X 0,Y 551.924,Z 1171.037,A -85,B 0,C 180,E1 19895.823,E2 19895.823} C_VEL
LIN {X 0,Y 551.905,Z 1173.7,A -85,B 0,C 180,E1 19893.22,E2 19893.22} C_VEL
LIN {X 0,Y 551.909,Z 1174.767,A -85,B 0,C 180,E1 19891.038,E2 19891.038} C_VEL
LIN {X 0,Y 551.911,Z 1174.766,A -85,B 0,C 180,E1 19888.858,E2 19888.858} C_VEL
LIN {X 0,Y 551.899,Z 1173.627,A -85,B 0,C 180,E1 19886.573,E2 19886.573} C_VEL
LIN {X 0,Y 551.941,Z 1170.693,A -85,B 0,C 180,E1 19883.865,E2 19883.865} C_VEL
LIN {X 0,Y 552.031,Z 1166.83,A -85,B 0,C 180,E1 19881.564,E2 19881.564} C_VEL
LIN {X 0,Y 552.198,Z 1161.994,A -85,B 0,C 180,E1 19879.357,E2 19879.357} C_VEL
LIN {X 0,Y 552.587,Z 1154.96,A -85,B 0,C 180,E1 19876.781,E2 19876.781} C_VEL
LIN {X 0,Y 553.22,Z 1145.953,A -85,B 0,C 180,E1 19874.163,E2 19874.163} C_VEL
LIN {X 0,Y 554.008,Z 1137.302,A -85,B 0,C 180,E1 19872.017,E2 19872.017} C_VEL
LIN {X 0,Y 555.258,Z 1125.879,A -85,B 0,C 180,E1 19869.553,E2 19869.553} C_VEL
LIN {X 0,Y 557.115,Z 1111.147,A -85,B 0,C 180,E1 19866.856,E2 19866.856} C_VEL
LIN {X 0,Y 559.318,Z 1096.65,A -85,B 0,C 180,E1 19864.48,E2 19864.48} C_VEL
LIN {X 0,Y 562,Z 1080.191,A -85,B 0,C 180,E1 19862.159,E2 19862.159} C_VEL
LIN {X 0,Y 564.615,Z 1065.204,A -85,B 0,C 180,E1 19860.274,E2 19860.274} C_VEL
LIN {X 0,Y 568.232,Z 1045.322,A -85,B 0,C 180,E1 19858.078,E2 19858.078} C_VEL
LIN {X 0,Y 571.39,Z 1028.027,A -85,B 0,C 180,E1 19856.405,E2 19856.405} C_VEL
LIN {X 0,Y 574.484,Z 1011.093,A -85,B 0,C 180,E1 19854.946,E2 19854.946} C_VEL
LIN {X 0,Y 578.288,Z 989.616,A -85,B 0,C 180,E1 19853.318,E2 19853.318} C_VEL
LIN {X 0,Y 581.564,Z 969.387,A -85,B 0,C 180,E1 19852.012,E2 19852.012} C_VEL
LIN {X 0,Y 584.482,Z 950.092,A -85,B 0,C 180,E1 19850.927,E2 19850.927} C_VEL
LIN {X 0,Y 587.71,Z 926.948,A -85,B 0,C 180,E1 19849.809,E2 19849.809} C_VEL
LIN {X 0,Y 590.587,Z 902.379,A -85,B 0,C 180,E1 19848.84,E2 19848.84} C_VEL
LIN {X 0,Y 592.767,Z 880.816,A -85,B 0,C 180,E1 19848.142,E2 19848.142} C_VEL
LIN {X 0,Y 594.939,Z 855.204,A -85,B 0,C 180,E1 19847.486,E2 19847.486} C_VEL
LIN {X 0,Y 596.365,Z 830.025,A -85,B 0,C 180,E1 19847.026,E2 19847.026} C_VEL
LIN {X 0,Y 602.551,Z 608.597,A -85,B 0,C 180,E1 19843.98,E2 19843.98} C_VEL
LIN {X 0,Y 607.324,Z 445.642,A -85,B 0,C 180,E1 19841.693,E2 19841.693} C_VEL
LIN {X 0,Y 602.329,Z 420.094,A -85,B 0,C 180,E1 19840.649,E2 19840.649} C_VEL
LIN {X 0,Y 589.665,Z 401.091,A -85,B 0,C 180,E1 19838.704,E2 19838.704} C_VEL
LIN {X 0,Y 580.931,Z 388.359,A -85,B 0,C 180,E1 19837.229,E2 19837.229} C_VEL
LIN {X 0,Y 575.058,Z 376.216,A -85,B 0,C 180,E1 19835.137,E2 19835.137} C_VEL
LIN {X 0,Y 568.797,Z 363.817,A -85,B 0,C 180,E1 19832.782,E2 19832.782} C_VEL
LIN {X 0,Y 563.834,Z 354.574,A -85,B 0,C 180,E1 19830.831,E2 19830.831} C_VEL
LIN {X 0,Y 561.089,Z 349.544,A -85,B 0,C 180,E1 19829.697,E2 19829.697} C_VEL
LIN {X 0,Y 558.707,Z 345.113,A -85,B 0,C 180,E1 19828.661,E2 19828.661} C_VEL
LIN {X 0,Y 556.779,Z 341.85,A -85,B 0,C 180,E1 19827.835,E2 19827.835} C_VEL
LIN {X 0,Y 555.922,Z 340.101,A -85,B 0,C 180,E1 19827.416,E2 19827.416} C_VEL
LIN {X 0,Y 553.79,Z 336.743,A -85,B 0,C 180,E1 19826.485,E2 19826.485} C_VEL
LIN {X 0,Y 553.506,Z 335.443,A -85,B 0,C 180,E1 19826.13,E2 19826.13} C_VEL
LIN {X 0,Y 553.472,Z 335.237,A -85,B 0,C 180,E1 19822.744,E2 19822.744} C_VEL
LIN {X 0,Y 553.493,Z 335.233,A -85,B 0,C 180,E1 19819.524,E2 19819.524} C_VEL
LIN {X 0,Y 553.482,Z 335.274,A -85,B 0,C 180,E1 19816.153,E2 19816.153} C_VEL
LIN {X 0,Y 553.492,Z 335.217,A -85,B 0,C 180,E1 19812.838,E2 19812.838} C_VEL
LIN {X 0,Y 553.494,Z 335.284,A -85,B 0,C 180,E1 19809.462,E2 19809.462} C_VEL
LIN {X 0,Y 553.482,Z 335.215,A -85,B 0,C 180,E1 19806.119,E2 19806.119} C_VEL
LIN {X 0,Y 553.492,Z 335.281,A -85,B 0,C 180,E1 19802.796,E2 19802.796} C_VEL
LIN {X 0,Y 553.481,Z 335.222,A -85,B 0,C 180,E1 19799.379,E2 19799.379} C_VEL
LIN {X 0,Y 553.496,Z 335.265,A -85,B 0,C 180,E1 19796.064,E2 19796.064} C_VEL
LIN {X 0,Y 553.47,Z 335.232,A -85,B 0,C 180,E1 19792.735,E2 19792.735} C_VEL
LIN {X 0,Y 553.483,Z 335.243,A -85,B 0,C 180,E1 19789.382,E2 19789.382} C_VEL
LIN {X 0,Y 553.502,Z 335.251,A -85,B 0,C 180,E1 19785.991,E2 19785.991} C_VEL
LIN {X 0,Y 553.453,Z 335.23,A -85,B 0,C 180,E1 19782.765,E2 19782.765} C_VEL
LIN {X 0,Y 553.505,Z 335.285,A -85,B 0,C 180,E1 19779.485,E2 19779.485} C_VEL
LIN {X 0,Y 553.449,Z 335.23,A -85,B 0,C 180,E1 19776.342,E2 19776.342} C_VEL
LIN {X 0,Y 553.558,Z 335.704,A -85,B 0,C 180,E1 19775.326,E2 19775.326} C_VEL
LIN {X 0,Y 555.045,Z 339.17,A -85,B 0,C 180,E1 19774.49,E2 19774.49} C_VEL
LIN {X 0,Y 556.619,Z 341.213,A -85,B 0,C 180,E1 19773.889,E2 19773.889} C_VEL
LIN {X 0,Y 558.708,Z 345.087,A -85,B 0,C 180,E1 19772.963,E2 19772.963} C_VEL
LIN {X 0,Y 559.885,Z 347.33,A -85,B 0,C 180,E1 19772.448,E2 19772.448} C_VEL
LIN {X 0,Y 562.447,Z 351.719,A -85,B 0,C 180,E1 19771.425,E2 19771.425} C_VEL
LIN {X 0,Y 565.508,Z 357.356,A -85,B 0,C 180,E1 19770.208,E2 19770.208} C_VEL
LIN {X 0,Y 567.375,Z 360.036,A -85,B 0,C 180,E1 19769.733,E2 19769.733} C_VEL
LIN {X 0,Y 577.189,Z 372.32,A -85,B 0,C 180,E1 19767.958,E2 19767.958} C_VEL
LIN {X 0,Y 586.001,Z 383.876,A -85,B 0,C 180,E1 19766.467,E2 19766.467} C_VEL
LIN {X 0,Y 596.846,Z 398.558,A -85,B 0,C 180,E1 19764.75,E2 19764.75} C_VEL
LIN {X 0,Y 610.394,Z 418.274,A -85,B 0,C 180,E1 19762.751,E2 19762.751} C_VEL
LIN {X 0,Y 612.101,Z 421.241,A -85,B 0,C 180,E1 19762.502,E2 19762.502} C_VEL
LIN {X 0,Y 605.521,Z 624.344,A -85,B 0,C 180,E1 19759.542,E2 19759.542} C_VEL
LIN {X 0,Y 599.392,Z 827.649,A -85,B 0,C 180,E1 19756.64,E2 19756.64} C_VEL
LIN {X 0,Y 597.71,Z 855.761,A -85,B 0,C 180,E1 19756.111,E2 19756.111} C_VEL
LIN {X 0,Y 595.618,Z 881.246,A -85,B 0,C 180,E1 19755.456,E2 19755.456} C_VEL
LIN {X 0,Y 593.598,Z 902.402,A -85,B 0,C 180,E1 19754.79,E2 19754.79} C_VEL
LIN {X 0,Y 591.286,Z 923.77,A -85,B 0,C 180,E1 19753.994,E2 19753.994} C_VEL
LIN {X 0,Y 588.323,Z 948.694,A -85,B 0,C 180,E1 19752.902,E2 19752.902} C_VEL
LIN {X 0,Y 584.914,Z 973.244,A -85,B 0,C 180,E1 19751.614,E2 19751.614} C_VEL
LIN {X 0,Y 582.046,Z 992.74,A -85,B 0,C 180,E1 19750.445,E2 19750.445} C_VEL
LIN {X 0,Y 579.161,Z 1011.405,A -85,B 0,C 180,E1 19749.188,E2 19749.188} C_VEL
LIN {X 0,Y 576.155,Z 1030.133,A -85,B 0,C 180,E1 19747.778,E2 19747.778} C_VEL
LIN {X 0,Y 572.776,Z 1049.353,A -85,B 0,C 180,E1 19746.113,E2 19746.113} C_VEL
LIN {X 0,Y 569.08,Z 1069.746,A -85,B 0,C 180,E1 19744.089,E2 19744.089} C_VEL
LIN {X 0,Y 566.114,Z 1086.365,A -85,B 0,C 180,E1 19742.235,E2 19742.235} C_VEL
LIN {X 0,Y 563.533,Z 1101.36,A -85,B 0,C 180,E1 19740.376,E2 19740.376} C_VEL
LIN {X 0,Y 560.657,Z 1118.746,A -85,B 0,C 180,E1 19737.971,E2 19737.971} C_VEL
LIN {X 0,Y 558.22,Z 1134.454,A -85,B 0,C 180,E1 19735.46,E2 19735.46} C_VEL
LIN {X 0,Y 556.504,Z 1146.564,A -85,B 0,C 180,E1 19733.283,E2 19733.283} C_VEL
LIN {X 0,Y 554.974,Z 1158.864,A -85,B 0,C 180,E1 19730.789,E2 19730.789} C_VEL
LIN {X 0,Y 553.727,Z 1170.678,A -85,B 0,C 180,E1 19727.985,E2 19727.985} C_VEL
LIN {X 0,Y 552.974,Z 1179.155,A -85,B 0,C 180,E1 19725.629,E2 19725.629} C_VEL
LIN {X 0,Y 552.5,Z 1186.376,A -85,B 0,C 180,E1 19723.287,E2 19723.287} C_VEL
LIN {X 0,Y 552.151,Z 1193.351,A -85,B 0,C 180,E1 19720.538,E2 19720.538} C_VEL
LIN {X 0,Y 551.982,Z 1198.733,A -85,B 0,C 180,E1 19717.703,E2 19717.703} C_VEL
LIN {X 0,Y 551.929,Z 1201.987,A -85,B 0,C 180,E1 19715.301,E2 19715.301} C_VEL
LIN {X 0,Y 551.915,Z 1204.047,A -85,B 0,C 180,E1 19712.907,E2 19712.907} C_VEL
LIN {X 0,Y 551.894,Z 1204.917,A -85,B 0,C 180,E1 19710.415,E2 19710.415} C_VEL
LIN {X 0,Y 551.908,Z 1204.318,A -85,B 0,C 180,E1 19707.508,E2 19707.508} C_VEL
LIN {X 0,Y 551.925,Z 1202.327,A -85,B 0,C 180,E1 19705.011,E2 19705.011} C_VEL
LIN {X 0,Y 551.977,Z 1199.211,A -85,B 0,C 180,E1 19702.61,E2 19702.61} C_VEL
LIN {X 0,Y 552.099,Z 1194.674,A -85,B 0,C 180,E1 19700.093,E2 19700.093} C_VEL
LIN {X 0,Y 552.426,Z 1187.587,A -85,B 0,C 180,E1 19697.136,E2 19697.136} C_VEL
LIN {X 0,Y 552.909,Z 1180.211,A -85,B 0,C 180,E1 19694.691,E2 19694.691} C_VEL
LIN {X 0,Y 553.56,Z 1172.297,A -85,B 0,C 180,E1 19692.443,E2 19692.443} C_VEL
LIN {X 0,Y 554.493,Z 1163.149,A -85,B 0,C 180,E1 19690.183,E2 19690.183} C_VEL
LIN {X 0,Y 556.012,Z 1150.58,A -85,B 0,C 180,E1 19687.478,E2 19687.478} C_VEL
LIN {X 0,Y 557.839,Z 1136.994,A -85,B 0,C 180,E1 19684.975,E2 19684.975} C_VEL
LIN {X 0,Y 559.757,Z 1124.371,A -85,B 0,C 180,E1 19682.903,E2 19682.903} C_VEL
LIN {X 0,Y 562.005,Z 1110.288,A -85,B 0,C 180,E1 19680.825,E2 19680.825} C_VEL
LIN {X 0,Y 565.269,Z 1091.453,A -85,B 0,C 180,E1 19678.368,E2 19678.368} C_VEL
LIN {X 0,Y 568.281,Z 1074.304,A -85,B 0,C 180,E1 19676.402,E2 19676.402} C_VEL
LIN {X 0,Y 571.112,Z 1058.483,A -85,B 0,C 180,E1 19674.769,E2 19674.769} C_VEL
LIN {X 0,Y 574.031,Z 1042.218,A -85,B 0,C 180,E1 19673.251,E2 19673.251} C_VEL
LIN {X 0,Y 576.443,Z 1028.342,A -85,B 0,C 180,E1 19672.083,E2 19672.083} C_VEL
LIN {X 0,Y 579.265,Z 1010.741,A -85,B 0,C 180,E1 19670.765,E2 19670.765} C_VEL
LIN {X 0,Y 582.146,Z 992.115,A -85,B 0,C 180,E1 19669.515,E2 19669.515} C_VEL
LIN {X 0,Y 585.352,Z 970.44,A -85,B 0,C 180,E1 19668.227,E2 19668.227} C_VEL
LIN {X 0,Y 588.849,Z 944.365,A -85,B 0,C 180,E1 19666.9,E2 19666.9} C_VEL
LIN {X 0,Y 591.36,Z 923.086,A -85,B 0,C 180,E1 19665.979,E2 19665.979} C_VEL
LIN {X 0,Y 593.608,Z 902.301,A -85,B 0,C 180,E1 19665.207,E2 19665.207} C_VEL
LIN {X 0,Y 595.639,Z 880.997,A -85,B 0,C 180,E1 19664.537,E2 19664.537} C_VEL
LIN {X 0,Y 597.713,Z 855.754,A -85,B 0,C 180,E1 19663.889,E2 19663.889} C_VEL
LIN {X 0,Y 599.376,Z 827.904,A -85,B 0,C 180,E1 19663.365,E2 19663.365} C_VEL
LIN {X 0,Y 602.005,Z 740.257,A -85,B 0,C 180,E1 19662.117,E2 19662.117} C_VEL
LIN {X 0,Y 608.797,Z 522.183,A -85,B 0,C 180,E1 19658.978,E2 19658.978} C_VEL
LIN {X 0,Y 611.969,Z 420.73,A -85,B 0,C 180,E1 19657.476,E2 19657.476} C_VEL
LIN {X 0,Y 598.428,Z 400.743,A -85,B 0,C 180,E1 19655.495,E2 19655.495} C_VEL
LIN {X 0,Y 586.608,Z 384.712,A -85,B 0,C 180,E1 19653.64,E2 19653.64} C_VEL
LIN {X 0,Y 579.253,Z 375.07,A -85,B 0,C 180,E1 19652.41,E2 19652.41} C_VEL
LIN {X 0,Y 571.269,Z 364.87,A -85,B 0,C 180,E1 19650.999,E2 19650.999} C_VEL
LIN {X 0,Y 566.03,Z 358.339,A -85,B 0,C 180,E1 19649.995,E2 19649.995} C_VEL
LIN {X 0,Y 564.173,Z 354.902,A -85,B 0,C 180,E1 19649.285,E2 19649.285} C_VEL
LIN {X 0,Y 561.337,Z 349.765,A -85,B 0,C 180,E1 19648.15,E2 19648.15} C_VEL
LIN {X 0,Y 558.652,Z 345.027,A -85,B 0,C 180,E1 19647.04,E2 19647.04} C_VEL
LIN {X 0,Y 556.582,Z 341.105,A -85,B 0,C 180,E1 19646.113,E2 19646.113} C_VEL
LIN {X 0,Y 553.879,Z 337.006,A -85,B 0,C 180,E1 19644.988,E2 19644.988} C_VEL
LIN {X 0,Y 553.522,Z 335.458,A -85,B 0,C 180,E1 19644.591,E2 19644.591} C_VEL
LIN {X 0,Y 553.45,Z 335.266,A -85,B 0,C 180,E1 19641.404,E2 19641.404} C_VEL
LIN {X 0,Y 553.498,Z 335.22,A -85,B 0,C 180,E1 19638.157,E2 19638.157} C_VEL
LIN {X 0,Y 553.47,Z 335.288,A -85,B 0,C 180,E1 19634.865,E2 19634.865} C_VEL
LIN {X 0,Y 553.467,Z 335.225,A -85,B 0,C 180,E1 19631.462,E2 19631.462} C_VEL
LIN {X 0,Y 553.499,Z 335.261,A -85,B 0,C 180,E1 19628.205,E2 19628.205} C_VEL
LIN {X 0,Y 553.467,Z 335.234,A -85,B 0,C 180,E1 19624.871,E2 19624.871} C_VEL
LIN {X 0,Y 553.496,Z 335.246,A -85,B 0,C 180,E1 19621.553,E2 19621.553} C_VEL
LIN {X 0,Y 553.493,Z 335.242,A -85,B 0,C 180,E1 19618.137,E2 19618.137} C_VEL
LIN {X 0,Y 553.477,Z 335.232,A -85,B 0,C 180,E1 19614.817,E2 19614.817} C_VEL
LIN {X 0,Y 553.494,Z 335.254,A -85,B 0,C 180,E1 19611.481,E2 19611.481} C_VEL
LIN {X 0,Y 553.489,Z 335.22,A -85,B 0,C 180,E1 19608.115,E2 19608.115} C_VEL
LIN {X 0,Y 553.494,Z 335.284,A -85,B 0,C 180,E1 19604.707,E2 19604.707} C_VEL
LIN {X 0,Y 553.478,Z 335.222,A -85,B 0,C 180,E1 19601.351,E2 19601.351} C_VEL
LIN {X 0,Y 553.492,Z 335.258,A -85,B 0,C 180,E1 19597.929,E2 19597.929} C_VEL
LIN {X 0,Y 553.498,Z 335.247,A -85,B 0,C 180,E1 19594.536,E2 19594.536} C_VEL
LIN {X 0,Y 553.541,Z 335.696,A -85,B 0,C 180,E1 19593.63,E2 19593.63} C_VEL
LIN {X 0,Y 555.091,Z 339.143,A -85,B 0,C 180,E1 19592.772,E2 19592.772} C_VEL
LIN {X 0,Y 556.438,Z 340.79,A -85,B 0,C 180,E1 19592.263,E2 19592.263} C_VEL
LIN {X 0,Y 558.146,Z 344.424,A -85,B 0,C 180,E1 19591.424,E2 19591.424} C_VEL
LIN {X 0,Y 559.447,Z 346.371,A -85,B 0,C 180,E1 19590.913,E2 19590.913} C_VEL
LIN {X 0,Y 562.323,Z 351.843,A -85,B 0,C 180,E1 19589.669,E2 19589.669} C_VEL
LIN {X 0,Y 564.89,Z 356.463,A -85,B 0,C 180,E1 19588.641,E2 19588.641} C_VEL
LIN {X 0,Y 570.085,Z 366.447,A -85,B 0,C 180,E1 19586.602,E2 19586.602} C_VEL
LIN {X 0,Y 576.246,Z 378.551,A -85,B 0,C 180,E1 19584.337,E2 19584.337} C_VEL
LIN {X 0,Y 581.515,Z 389.331,A -85,B 0,C 180,E1 19582.536,E2 19582.536} C_VEL
LIN {X 0,Y 594.54,Z 408.235,A -85,B 0,C 180,E1 19580.433,E2 19580.433} C_VEL
LIN {X 0,Y 602.555,Z 420.665,A -85,B 0,C 180,E1 19579.217,E2 19579.217} C_VEL
LIN {X 0,Y 607.343,Z 446.701,A -85,B 0,C 180,E1 19578.191,E2 19578.191} C_VEL
LIN {X 0,Y 600.49,Z 681.941,A -85,B 0,C 180,E1 19574.92,E2 19574.92} C_VEL
LIN {X 0,Y 599.552,Z 716.236,A -85,B 0,C 180,E1 19574.451,E2 19574.451} C_VEL
LIN {X 0,Y 598.639,Z 723.943,A -85,B 0,C 180,E1 19574.417,E2 19574.417} C_VEL
LIN {X 0,Y 593.777,Z 744.565,A -85,B 0,C 180,E1 19574.573,E2 19574.573} C_VEL
LIN {X 0,Y 593.086,Z 751.174,A -85,B 0,C 180,E1 19574.534,E2 19574.534} C_VEL
LIN {X 0,Y 590.641,Z 832.233,A -85,B 0,C 180,E1 19573.403,E2 19573.403} C_VEL
LIN {X 0,Y 588.804,Z 860.328,A -85,B 0,C 180,E1 19572.857,E2 19572.857} C_VEL
LIN {X 0,Y 586.818,Z 882.722,A -85,B 0,C 180,E1 19572.261,E2 19572.261} C_VEL
LIN {X 0,Y 584.534,Z 904.306,A -85,B 0,C 180,E1 19571.55,E2 19571.55} C_VEL
LIN {X 0,Y 581.229,Z 930.6,A -85,B 0,C 180,E1 19570.479,E2 19570.479} C_VEL
LIN {X 0,Y 578.219,Z 951.406,A -85,B 0,C 180,E1 19569.457,E2 19569.457} C_VEL
LIN {X 0,Y 575.047,Z 971.597,A -85,B 0,C 180,E1 19568.307,E2 19568.307} C_VEL
LIN {X 0,Y 571.005,Z 995.247,A -85,B 0,C 180,E1 19566.727,E2 19566.727} C_VEL
LIN {X 0,Y 567.807,Z 1012.668,A -85,B 0,C 180,E1 19565.38,E2 19565.38} C_VEL
LIN {X 0,Y 564.697,Z 1028.921,A -85,B 0,C 180,E1 19563.962,E2 19563.962} C_VEL
LIN {X 0,Y 561.131,Z 1047.517,A -85,B 0,C 180,E1 19562.134,E2 19562.134} C_VEL
LIN {X 0,Y 557.49,Z 1066.107,A -85,B 0,C 180,E1 19560.026,E2 19560.026} C_VEL
LIN {X 0,Y 554.801,Z 1080.607,A -85,B 0,C 180,E1 19558.176,E2 19558.176} C_VEL
LIN {X 0,Y 552.016,Z 1096.622,A -85,B 0,C 180,E1 19555.883,E2 19555.883} C_VEL
LIN {X 0,Y 549.631,Z 1111.126,A -85,B 0,C 180,E1 19553.478,E2 19553.478} C_VEL
LIN {X 0,Y 547.925,Z 1122.795,A -85,B 0,C 180,E1 19551.294,E2 19551.294} C_VEL
LIN {X 0,Y 546.351,Z 1135.624,A -85,B 0,C 180,E1 19548.557,E2 19548.557} C_VEL
LIN {X 0,Y 545.429,Z 1144.8,A -85,B 0,C 180,E1 19546.289,E2 19546.289} C_VEL
LIN {X 0,Y 544.804,Z 1152.358,A -85,B 0,C 180,E1 19544.129,E2 19544.129} C_VEL
LIN {X 0,Y 544.323,Z 1159.978,A -85,B 0,C 180,E1 19541.55,E2 19541.55} C_VEL
LIN {X 0,Y 544.063,Z 1166.033,A -85,B 0,C 180,E1 19538.881,E2 19538.881} C_VEL
LIN {X 0,Y 543.952,Z 1169.758,A -85,B 0,C 180,E1 19536.756,E2 19536.756} C_VEL
LIN {X 0,Y 543.906,Z 1172.58,A -85,B 0,C 180,E1 19534.534,E2 19534.534} C_VEL
LIN {X 0,Y 543.907,Z 1174.577,A -85,B 0,C 180,E1 19531.896,E2 19531.896} C_VEL
LIN {X 0,Y 543.895,Z 1174.878,A -85,B 0,C 180,E1 19529.368,E2 19529.368} C_VEL
LIN {X 0,Y 543.907,Z 1174.034,A -85,B 0,C 180,E1 19527.155,E2 19527.155} C_VEL
LIN {X 0,Y 543.913,Z 1172.224,A -85,B 0,C 180,E1 19525.044,E2 19525.044} C_VEL
LIN {X 0,Y 543.977,Z 1169.096,A -85,B 0,C 180,E1 19522.714,E2 19522.714} C_VEL
LIN {X 0,Y 544.133,Z 1163.772,A -85,B 0,C 180,E1 19519.947,E2 19519.947} C_VEL
LIN {X 0,Y 544.447,Z 1157.806,A -85,B 0,C 180,E1 19517.592,E2 19517.592} C_VEL
LIN {X 0,Y 544.882,Z 1151.241,A -85,B 0,C 180,E1 19515.44,E2 19515.44} C_VEL
LIN {X 0,Y 545.671,Z 1142.298,A -85,B 0,C 180,E1 19512.952,E2 19512.952} C_VEL
LIN {X 0,Y 546.985,Z 1130.089,A -85,B 0,C 180,E1 19510.123,E2 19510.123} C_VEL
LIN {X 0,Y 548.829,Z 1116.54,A -85,B 0,C 180,E1 19507.393,E2 19507.393} C_VEL
LIN {X 0,Y 550.984,Z 1102.575,A -85,B 0,C 180,E1 19504.987,E2 19504.987} C_VEL
LIN {X 0,Y 553.288,Z 1089.037,A -85,B 0,C 180,E1 19502.909,E2 19502.909} C_VEL
LIN {X 0,Y 556.555,Z 1071.236,A -85,B 0,C 180,E1 19500.511,E2 19500.511} C_VEL
LIN {X 0,Y 559.61,Z 1055.078,A -85,B 0,C 180,E1 19498.605,E2 19498.605} C_VEL
LIN {X 0,Y 562.896,Z 1038.225,A -85,B 0,C 180,E1 19496.832,E2 19496.832} C_VEL
LIN {X 0,Y 566.965,Z 1017.215,A -85,B 0,C 180,E1 19494.906,E2 19494.906} C_VEL
LIN {X 0,Y 570.168,Z 999.857,A -85,B 0,C 180,E1 19493.524,E2 19493.524} C_VEL
LIN {X 0,Y 573.199,Z 982.626,A -85,B 0,C 180,E1 19492.309,E2 19492.309} C_VEL
LIN {X 0,Y 576.59,Z 962.312,A -85,B 0,C 180,E1 19491.052,E2 19491.052} C_VEL
LIN {X 0,Y 580.175,Z 938.399,A -85,B 0,C 180,E1 19489.797,E2 19489.797} C_VEL
LIN {X 0,Y 582.815,Z 918.732,A -85,B 0,C 180,E1 19488.923,E2 19488.923} C_VEL
LIN {X 0,Y 585.065,Z 899.791,A -85,B 0,C 180,E1 19488.202,E2 19488.202} C_VEL
LIN {X 0,Y 587.359,Z 877.711,A -85,B 0,C 180,E1 19487.503,E2 19487.503} C_VEL
LIN {X 0,Y 589.528,Z 851.285,A -85,B 0,C 180,E1 19486.857,E2 19486.857} C_VEL
LIN {X 0,Y 590.794,Z 829.003,A -85,B 0,C 180,E1 19486.456,E2 19486.456} C_VEL
LIN {X 0,Y 597.457,Z 600.888,A -85,B 0,C 180,E1 19483.298,E2 19483.298} C_VEL
LIN {X 0,Y 602.15,Z 447.492,A -85,B 0,C 180,E1 19481.126,E2 19481.126} C_VEL
LIN {X 0,Y 597.831,Z 425.005,A -85,B 0,C 180,E1 19480.195,E2 19480.195} C_VEL
LIN {X 0,Y 585.337,Z 406.177,A -85,B 0,C 180,E1 19478.229,E2 19478.229} C_VEL
LIN {X 0,Y 572.708,Z 387.889,A -85,B 0,C 180,E1 19476.042,E2 19476.042} C_VEL
LIN {X 0,Y 566.011,Z 374.446,A -85,B 0,C 180,E1 19473.569,E2 19473.569} C_VEL
LIN {X 0,Y 560.704,Z 364.377,A -85,B 0,C 180,E1 19471.5,E2 19471.5} C_VEL
LIN {X 0,Y 558.698,Z 360.522,A -85,B 0,C 180,E1 19470.668,E2 19470.668} C_VEL
LIN {X 0,Y 555.829,Z 355.278,A -85,B 0,C 180,E1 19469.465,E2 19469.465} C_VEL
LIN {X 0,Y 553.61,Z 351.114,A -85,B 0,C 180,E1 19468.478,E2 19468.478} C_VEL
LIN {X 0,Y 551.576,Z 347.267,A -85,B 0,C 180,E1 19467.533,E2 19467.533} C_VEL
LIN {X 0,Y 548.802,Z 342.673,A -85,B 0,C 180,E1 19466.279,E2 19466.279} C_VEL
LIN {X 0,Y 547.966,Z 341.086,A -85,B 0,C 180,E1 19465.856,E2 19465.856} C_VEL
LIN {X 0,Y 545.803,Z 337.524,A -85,B 0,C 180,E1 19464.804,E2 19464.804} C_VEL
LIN {X 0,Y 545.556,Z 336.443,A -85,B 0,C 180,E1 19464.47,E2 19464.47} C_VEL
LIN {X 0,Y 545.564,Z 336.269,A -85,B 0,C 180,E1 19461.39,E2 19461.39} C_VEL
LIN {X 0,Y 545.547,Z 336.209,A -85,B 0,C 180,E1 19457.934,E2 19457.934} C_VEL
LIN {X 0,Y 545.542,Z 336.245,A -85,B 0,C 180,E1 19454.543,E2 19454.543} C_VEL
LIN {X 0,Y 545.549,Z 336.22,A -85,B 0,C 180,E1 19451.203,E2 19451.203} C_VEL
LIN {X 0,Y 545.551,Z 336.221,A -85,B 0,C 180,E1 19447.901,E2 19447.901} C_VEL
LIN {X 0,Y 545.553,Z 336.241,A -85,B 0,C 180,E1 19444.415,E2 19444.415} C_VEL
LIN {X 0,Y 545.536,Z 336.21,A -85,B 0,C 180,E1 19441.05,E2 19441.05} C_VEL
LIN {X 0,Y 545.558,Z 336.263,A -85,B 0,C 180,E1 19437.689,E2 19437.689} C_VEL
LIN {X 0,Y 545.553,Z 336.204,A -85,B 0,C 180,E1 19434.32,E2 19434.32} C_VEL
LIN {X 0,Y 545.532,Z 336.277,A -85,B 0,C 180,E1 19430.931,E2 19430.931} C_VEL
LIN {X 0,Y 545.551,Z 336.204,A -85,B 0,C 180,E1 19427.51,E2 19427.51} C_VEL
LIN {X 0,Y 545.547,Z 336.255,A -85,B 0,C 180,E1 19424.199,E2 19424.199} C_VEL
LIN {X 0,Y 545.516,Z 336.226,A -85,B 0,C 180,E1 19420.847,E2 19420.847} C_VEL
LIN {X 0,Y 545.566,Z 336.216,A -85,B 0,C 180,E1 19417.591,E2 19417.591} C_VEL
LIN {X 0,Y 545.606,Z 336.781,A -85,B 0,C 180,E1 19416.967,E2 19416.967} C_VEL
LIN {X 0,Y 547.157,Z 340.147,A -85,B 0,C 180,E1 19416.066,E2 19416.066} C_VEL
LIN {X 0,Y 548.737,Z 342.275,A -85,B 0,C 180,E1 19415.401,E2 19415.401} C_VEL
LIN {X 0,Y 550.573,Z 345.86,A -85,B 0,C 180,E1 19414.499,E2 19414.499} C_VEL
LIN {X 0,Y 551.832,Z 347.668,A -85,B 0,C 180,E1 19413.989,E2 19413.989} C_VEL
LIN {X 0,Y 553.942,Z 351.445,A -85,B 0,C 180,E1 19413.059,E2 19413.059} C_VEL
LIN {X 0,Y 557.374,Z 357.624,A -85,B 0,C 180,E1 19411.615,E2 19411.615} C_VEL
LIN {X 0,Y 558.929,Z 360.301,A -85,B 0,C 180,E1 19411.117,E2 19411.117} C_VEL
LIN {X 0,Y 565.898,Z 368.72,A -85,B 0,C 180,E1 19409.763,E2 19409.763} C_VEL
LIN {X 0,Y 574.212,Z 379.211,A -85,B 0,C 180,E1 19408.243,E2 19408.243} C_VEL
LIN {X 0,Y 586.16,Z 394.957,A -85,B 0,C 180,E1 19406.213,E2 19406.213} C_VEL
LIN {X 0,Y 598.751,Z 412.82,A -85,B 0,C 180,E1 19404.233,E2 19404.233} C_VEL
LIN {X 0,Y 606.87,Z 425.04,A -85,B 0,C 180,E1 19403.03,E2 19403.03} C_VEL
LIN {X 0,Y 599.957,Z 628.414,A -85,B 0,C 180,E1 19400.045,E2 19400.045} C_VEL
LIN {X 0,Y 593.527,Z 827.1,A -85,B 0,C 180,E1 19397.171,E2 19397.171} C_VEL
LIN {X 0,Y 591.831,Z 854.691,A -85,B 0,C 180,E1 19396.654,E2 19396.654} C_VEL
LIN {X 0,Y 589.605,Z 880.745,A -85,B 0,C 180,E1 19395.983,E2 19395.983} C_VEL
LIN {X 0,Y 587.493,Z 901.917,A -85,B 0,C 180,E1 19395.315,E2 19395.315} C_VEL
LIN {X 0,Y 585.116,Z 923.017,A -85,B 0,C 180,E1 19394.526,E2 19394.526} C_VEL
LIN {X 0,Y 582.277,Z 946.02,A -85,B 0,C 180,E1 19393.518,E2 19393.518} C_VEL
LIN {X 0,Y 578.565,Z 972.445,A -85,B 0,C 180,E1 19392.148,E2 19392.148} C_VEL
LIN {X 0,Y 575.591,Z 991.911,A -85,B 0,C 180,E1 19390.977,E2 19390.977} C_VEL
LIN {X 0,Y 572.742,Z 1009.593,A -85,B 0,C 180,E1 19389.785,E2 19389.785} C_VEL
LIN {X 0,Y 569.806,Z 1027.081,A -85,B 0,C 180,E1 19388.473,E2 19388.473} C_VEL
LIN {X 0,Y 566.738,Z 1044.908,A -85,B 0,C 180,E1 19386.985,E2 19386.985} C_VEL
LIN {X 0,Y 564.183,Z 1059.043,A -85,B 0,C 180,E1 19385.667,E2 19385.667} C_VEL
LIN {X 0,Y 560.906,Z 1076.537,A -85,B 0,C 180,E1 19383.828,E2 19383.828} C_VEL
LIN {X 0,Y 557.047,Z 1097.132,A -85,B 0,C 180,E1 19381.368,E2 19381.368} C_VEL
LIN {X 0,Y 554.403,Z 1111.831,A -85,B 0,C 180,E1 19379.377,E2 19379.377} C_VEL
LIN {X 0,Y 552.178,Z 1125.071,A -85,B 0,C 180,E1 19377.383,E2 19377.383} C_VEL
LIN {X 0,Y 549.979,Z 1138.896,A -85,B 0,C 180,E1 19375.062,E2 19375.062} C_VEL
LIN {X 0,Y 547.868,Z 1153.714,A -85,B 0,C 180,E1 19372.196,E2 19372.196} C_VEL
LIN {X 0,Y 546.578,Z 1164.063,A -85,B 0,C 180,E1 19369.892,E2 19369.892} C_VEL
LIN {X 0,Y 545.61,Z 1173.107,A -85,B 0,C 180,E1 19367.6,E2 19367.6} C_VEL
LIN {X 0,Y 544.863,Z 1181.98,A -85,B 0,C 180,E1 19364.996,E2 19364.996} C_VEL
LIN {X 0,Y 544.318,Z 1190.062,A -85,B 0,C 180,E1 19362.088,E2 19362.088} C_VEL
LIN {X 0,Y 544.084,Z 1195.498,A -85,B 0,C 180,E1 19359.627,E2 19359.627} C_VEL
LIN {X 0,Y 543.976,Z 1199.529,A -85,B 0,C 180,E1 19357.286,E2 19357.286} C_VEL
LIN {X 0,Y 543.919,Z 1202.666,A -85,B 0,C 180,E1 19354.745,E2 19354.745} C_VEL
LIN {X 0,Y 543.91,Z 1204.6,A -85,B 0,C 180,E1 19351.896,E2 19351.896} C_VEL
LIN {X 0,Y 543.895,Z 1204.872,A -85,B 0,C 180,E1 19349.368,E2 19349.368} C_VEL
LIN {X 0,Y 543.915,Z 1204.043,A -85,B 0,C 180,E1 19347.049,E2 19347.049} C_VEL
LIN {X 0,Y 543.93,Z 1202.096,A -85,B 0,C 180,E1 19344.726,E2 19344.726} C_VEL
LIN {X 0,Y 543.983,Z 1198.889,A -85,B 0,C 180,E1 19342.289,E2 19342.289} C_VEL
LIN {X 0,Y 544.154,Z 1193.818,A -85,B 0,C 180,E1 19339.519,E2 19339.519} C_VEL
LIN {X 0,Y 544.53,Z 1186.674,A -85,B 0,C 180,E1 19336.622,E2 19336.622} C_VEL
LIN {X 0,Y 545.028,Z 1179.504,A -85,B 0,C 180,E1 19334.246,E2 19334.246} C_VEL
LIN {X 0,Y 545.784,Z 1171.461,A -85,B 0,C 180,E1 19331.957,E2 19331.957} C_VEL
LIN {X 0,Y 547.03,Z 1160.374,A -85,B 0,C 180,E1 19329.231,E2 19329.231} C_VEL
LIN {X 0,Y 548.681,Z 1147.711,A -85,B 0,C 180,E1 19326.592,E2 19326.592} C_VEL
LIN {X 0,Y 550.465,Z 1135.722,A -85,B 0,C 180,E1 19324.386,E2 19324.386} C_VEL
LIN {X 0,Y 552.553,Z 1122.681,A -85,B 0,C 180,E1 19322.238,E2 19322.238} C_VEL
LIN {X 0,Y 555.576,Z 1105.58,A -85,B 0,C 180,E1 19319.74,E2 19319.74} C_VEL
LIN {X 0,Y 558.687,Z 1088.211,A -85,B 0,C 180,E1 19317.526,E2 19317.526} C_VEL
LIN {X 0,Y 561.578,Z 1072.782,A -85,B 0,C 180,E1 19315.762,E2 19315.762} C_VEL
LIN {X 0,Y 564.69,Z 1056.261,A -85,B 0,C 180,E1 19314.057,E2 19314.057} C_VEL
LIN {X 0,Y 567.596,Z 1039.844,A -85,B 0,C 180,E1 19312.573,E2 19312.573} C_VEL
LIN {X 0,Y 571.593,Z 1016.529,A -85,B 0,C 180,E1 19310.71,E2 19310.71} C_VEL
LIN {X 0,Y 575.041,Z 995.274,A -85,B 0,C 180,E1 19309.238,E2 19309.238} C_VEL
LIN {X 0,Y 577.984,Z 976.172,A -85,B 0,C 180,E1 19308.064,E2 19308.064} C_VEL
LIN {X 0,Y 580.899,Z 955.802,A -85,B 0,C 180,E1 19306.962,E2 19306.962} C_VEL
LIN {X 0,Y 584.333,Z 930.001,A -85,B 0,C 180,E1 19305.756,E2 19305.756} C_VEL
LIN {X 0,Y 587.169,Z 904.973,A -85,B 0,C 180,E1 19304.791,E2 19304.791} C_VEL
LIN {X 0,Y 589.337,Z 883.428,A -85,B 0,C 180,E1 19304.094,E2 19304.094} C_VEL
LIN {X 0,Y 591.223,Z 861.848,A -85,B 0,C 180,E1 19303.518,E2 19303.518} C_VEL
LIN {X 0,Y 592.994,Z 837.269,A -85,B 0,C 180,E1 19302.999,E2 19302.999} C_VEL
LIN {X 0,Y 594.534,Z 799.87,A -85,B 0,C 180,E1 19302.424,E2 19302.424} C_VEL
LIN {X 0,Y 601.685,Z 576.694,A -85,B 0,C 180,E1 19299.202,E2 19299.202} C_VEL
LIN {X 0,Y 606.797,Z 424.784,A -85,B 0,C 180,E1 19296.96,E2 19296.96} C_VEL
LIN {X 0,Y 593.42,Z 405.09,A -85,B 0,C 180,E1 19294.952,E2 19294.952} C_VEL
LIN {X 0,Y 580.774,Z 387.734,A -85,B 0,C 180,E1 19292.901,E2 19292.901} C_VEL
LIN {X 0,Y 568.711,Z 372.14,A -85,B 0,C 180,E1 19290.772,E2 19290.772} C_VEL
LIN {X 0,Y 559.316,Z 360.765,A -85,B 0,C 180,E1 19288.978,E2 19288.978} C_VEL
LIN {X 0,Y 557.543,Z 358.086,A -85,B 0,C 180,E1 19288.492,E2 19288.492} C_VEL
LIN {X 0,Y 556.307,Z 355.797,A -85,B 0,C 180,E1 19287.977,E2 19287.977} C_VEL
LIN {X 0,Y 553.6,Z 351.038,A -85,B 0,C 180,E1 19286.843,E2 19286.843} C_VEL
LIN {X 0,Y 551.049,Z 346.397,A -85,B 0,C 180,E1 19285.701,E2 19285.701} C_VEL
LIN {X 0,Y 548.948,Z 342.937,A -85,B 0,C 180,E1 19284.768,E2 19284.768} C_VEL
LIN {X 0,Y 548.15,Z 341.234,A -85,B 0,C 180,E1 19284.346,E2 19284.346} C_VEL
LIN {X 0,Y 546.021,Z 338.215,A -85,B 0,C 180,E1 19283.414,E2 19283.414} C_VEL
LIN {X 0,Y 545.551,Z 336.43,A -85,B 0,C 180,E1 19282.922,E2 19282.922} C_VEL
LIN {X 0,Y 545.52,Z 336.239,A -85,B 0,C 180,E1 19279.591,E2 19279.591} C_VEL
LIN {X 0,Y 545.563,Z 336.234,A -85,B 0,C 180,E1 19276.285,E2 19276.285} C_VEL
LIN {X 0,Y 545.519,Z 336.216,A -85,B 0,C 180,E1 19273.029,E2 19273.029} C_VEL
LIN {X 0,Y 545.547,Z 336.268,A -85,B 0,C 180,E1 19269.582,E2 19269.582} C_VEL
LIN {X 0,Y 545.556,Z 336.201,A -85,B 0,C 180,E1 19266.208,E2 19266.208} C_VEL
LIN {X 0,Y 545.538,Z 336.279,A -85,B 0,C 180,E1 19262.837,E2 19262.837} C_VEL
LIN {X 0,Y 545.556,Z 336.201,A -85,B 0,C 180,E1 19259.475,E2 19259.475} C_VEL
LIN {X 0,Y 545.556,Z 336.262,A -85,B 0,C 180,E1 19256.006,E2 19256.006} C_VEL
LIN {X 0,Y 545.54,Z 336.207,A -85,B 0,C 180,E1 19252.629,E2 19252.629} C_VEL
LIN {X 0,Y 545.555,Z 336.238,A -85,B 0,C 180,E1 19249.332,E2 19249.332} C_VEL
LIN {X 0,Y 545.548,Z 336.226,A -85,B 0,C 180,E1 19245.891,E2 19245.891} C_VEL
LIN {X 0,Y 545.551,Z 336.218,A -85,B 0,C 180,E1 19242.617,E2 19242.617} C_VEL
LIN {X 0,Y 545.544,Z 336.26,A -85,B 0,C 180,E1 19239.284,E2 19239.284} C_VEL
LIN {X 0,Y 545.544,Z 336.211,A -85,B 0,C 180,E1 19235.875,E2 19235.875} C_VEL
LIN {X 0,Y 545.615,Z 336.747,A -85,B 0,C 180,E1 19235.261,E2 19235.261} C_VEL
LIN {X 0,Y 547.429,Z 340.47,A -85,B 0,C 180,E1 19234.233,E2 19234.233} C_VEL
LIN {X 0,Y 548.631,Z 342.155,A -85,B 0,C 180,E1 19233.713,E2 19233.713} C_VEL
LIN {X 0,Y 550.566,Z 345.808,A -85,B 0,C 180,E1 19232.764,E2 19232.764} C_VEL
LIN {X 0,Y 551.566,Z 347.262,A -85,B 0,C 180,E1 19232.349,E2 19232.349} C_VEL
LIN {X 0,Y 553.612,Z 351.11,A -85,B 0,C 180,E1 19231.404,E2 19231.404} C_VEL
LIN {X 0,Y 557.213,Z 357.777,A -85,B 0,C 180,E1 19229.838,E2 19229.838} C_VEL
LIN {X 0,Y 560.209,Z 363.452,A -85,B 0,C 180,E1 19228.589,E2 19228.589} C_VEL
LIN {X 0,Y 564.481,Z 371.471,A -85,B 0,C 180,E1 19226.913,E2 19226.913} C_VEL
LIN {X 0,Y 570.987,Z 384.525,A -85,B 0,C 180,E1 19224.452,E2 19224.452} C_VEL
LIN {X 0,Y 573.296,Z 388.94,A -85,B 0,C 180,E1 19223.723,E2 19223.723} C_VEL
LIN {X 0,Y 585.828,Z 406.922,A -85,B 0,C 180,E1 19221.59,E2 19221.59} C_VEL
LIN {X 0,Y 597.958,Z 425.252,A -85,B 0,C 180,E1 19219.688,E2 19219.688} C_VEL
LIN {X 0,Y 602.193,Z 448.582,A -85,B 0,C 180,E1 19218.753,E2 19218.753} C_VEL
LIN {X 0,Y 595.024,Z 683.174,A -85,B 0,C 180,E1 19215.47,E2 19215.47} C_VEL
LIN {X 0,Y 593.086,Z 751.174,A -85,B 0,C 180,E1 19214.534,E2 19214.534} C_VEL
LIN {X 0,Y 592.19,Z 758.88,A -85,B 0,C 180,E1 19214.498,E2 19214.498} C_VEL
LIN {X 0,Y 587.298,Z 779.496,A -85,B 0,C 180,E1 19214.66,E2 19214.66} C_VEL
LIN {X 0,Y 586.604,Z 786.106,A -85,B 0,C 180,E1 19214.622,E2 19214.622} C_VEL
LIN {X 0,Y 584.928,Z 835.354,A -85,B 0,C 180,E1 19213.917,E2 19213.917} C_VEL
LIN {X 0,Y 583.016,Z 861.982,A -85,B 0,C 180,E1 19213.378,E2 19213.378} C_VEL
LIN {X 0,Y 581.008,Z 883.684,A -85,B 0,C 180,E1 19212.792,E2 19212.792} C_VEL
LIN {X 0,Y 578.376,Z 907.525,A -85,B 0,C 180,E1 19211.993,E2 19211.993} C_VEL
LIN {X 0,Y 575.063,Z 932.23,A -85,B 0,C 180,E1 19210.958,E2 19210.958} C_VEL
LIN {X 0,Y 572.057,Z 952.19,A -85,B 0,C 180,E1 19209.967,E2 19209.967} C_VEL
LIN {X 0,Y 568.623,Z 973.232,A -85,B 0,C 180,E1 19208.756,E2 19208.756} C_VEL
LIN {X 0,Y 564.553,Z 995.96,A -85,B 0,C 180,E1 19207.217,E2 19207.217} C_VEL
LIN {X 0,Y 561.18,Z 1013.702,A -85,B 0,C 180,E1 19205.835,E2 19205.835} C_VEL
LIN {X 0,Y 557.897,Z 1030.371,A -85,B 0,C 180,E1 19204.371,E2 19204.371} C_VEL
LIN {X 0,Y 554.082,Z 1049.411,A -85,B 0,C 180,E1 19202.47,E2 19202.47} C_VEL
LIN {X 0,Y 550.452,Z 1066.876,A -85,B 0,C 180,E1 19200.451,E2 19200.451} C_VEL
LIN {X 0,Y 547.443,Z 1082.073,A -85,B 0,C 180,E1 19198.471,E2 19198.471} C_VEL
LIN {X 0,Y 544.239,Z 1099.223,A -85,B 0,C 180,E1 19195.929,E2 19195.929} C_VEL
LIN {X 0,Y 541.992,Z 1112.222,A -85,B 0,C 180,E1 19193.714,E2 19193.714} C_VEL
LIN {X 0,Y 540.04,Z 1124.895,A -85,B 0,C 180,E1 19191.278,E2 19191.278} C_VEL
LIN {X 0,Y 538.449,Z 1136.698,A -85,B 0,C 180,E1 19188.627,E2 19188.627} C_VEL
LIN {X 0,Y 537.354,Z 1146.825,A -85,B 0,C 180,E1 19185.985,E2 19185.985} C_VEL
LIN {X 0,Y 536.613,Z 1156.039,A -85,B 0,C 180,E1 19183.14,E2 19183.14} C_VEL
LIN {X 0,Y 536.244,Z 1162.035,A -85,B 0,C 180,E1 19180.855,E2 19180.855} C_VEL
LIN {X 0,Y 536.049,Z 1166.862,A -85,B 0,C 180,E1 19178.582,E2 19178.582} C_VEL
LIN {X 0,Y 535.935,Z 1171.04,A -85,B 0,C 180,E1 19175.997,E2 19175.997} C_VEL
LIN {X 0,Y 535.903,Z 1173.7,A -85,B 0,C 180,E1 19173.316,E2 19173.316} C_VEL
LIN {X 0,Y 535.909,Z 1174.767,A -85,B 0,C 180,E1 19171.069,E2 19171.069} C_VEL
LIN {X 0,Y 535.909,Z 1174.788,A -85,B 0,C 180,E1 19168.931,E2 19168.931} C_VEL
LIN {X 0,Y 535.902,Z 1173.761,A -85,B 0,C 180,E1 19166.684,E2 19166.684} C_VEL
LIN {X 0,Y 535.938,Z 1171.078,A -85,B 0,C 180,E1 19163.942,E2 19163.942} C_VEL
LIN {X 0,Y 536.044,Z 1166.901,A -85,B 0,C 180,E1 19161.349,E2 19161.349} C_VEL
LIN {X 0,Y 536.234,Z 1162.245,A -85,B 0,C 180,E1 19159.145,E2 19159.145} C_VEL
LIN {X 0,Y 536.617,Z 1155.984,A -85,B 0,C 180,E1 19156.751,E2 19156.751} C_VEL
LIN {X 0,Y 537.358,Z 1146.757,A -85,B 0,C 180,E1 19153.904,E2 19153.904} C_VEL
LIN {X 0,Y 538.4,Z 1137.052,A -85,B 0,C 180,E1 19151.372,E2 19151.372} C_VEL
LIN {X 0,Y 539.976,Z 1125.333,A -85,B 0,C 180,E1 19148.72,E2 19148.72} C_VEL
LIN {X 0,Y 541.969,Z 1112.34,A -85,B 0,C 180,E1 19146.218,E2 19146.218} C_VEL
LIN {X 0,Y 544.134,Z 1099.741,A -85,B 0,C 180,E1 19144.066,E2 19144.066} C_VEL
LIN {X 0,Y 547.398,Z 1082.334,A -85,B 0,C 180,E1 19141.475,E2 19141.475} C_VEL
LIN {X 0,Y 550.315,Z 1067.531,A -85,B 0,C 180,E1 19139.541,E2 19139.541} C_VEL
LIN {X 0,Y 553.809,Z 1050.617,A -85,B 0,C 180,E1 19137.574,E2 19137.574} C_VEL
LIN {X 0,Y 557.736,Z 1031.236,A -85,B 0,C 180,E1 19135.618,E2 19135.618} C_VEL
LIN {X 0,Y 561.107,Z 1014.108,A -85,B 0,C 180,E1 19134.108,E2 19134.108} C_VEL
LIN {X 0,Y 564.365,Z 996.998,A -85,B 0,C 180,E1 19132.769,E2 19132.769} C_VEL
LIN {X 0,Y 568.3,Z 975.366,A -85,B 0,C 180,E1 19131.283,E2 19131.283} C_VEL
LIN {X 0,Y 572.002,Z 952.592,A -85,B 0,C 180,E1 19129.964,E2 19129.964} C_VEL
LIN {X 0,Y 574.997,Z 932.788,A -85,B 0,C 180,E1 19128.978,E2 19128.978} C_VEL
LIN {X 0,Y 578.25,Z 908.828,A -85,B 0,C 180,E1 19127.963,E2 19127.963} C_VEL
LIN {X 0,Y 580.984,Z 884.025,A -85,B 0,C 180,E1 19127.126,E2 19127.126} C_VEL
LIN {X 0,Y 583.006,Z 862.33,A -85,B 0,C 180,E1 19126.54,E2 19126.54} C_VEL
LIN {X 0,Y 584.912,Z 836.01,A -85,B 0,C 180,E1 19126.001,E2 19126.001} C_VEL
LIN {X 0,Y 586.552,Z 788.406,A -85,B 0,C 180,E1 19125.318,E2 19125.318} C_VEL
LIN {X 0,Y 593.402,Z 562.333,A -85,B 0,C 180,E1 19122.168,E2 19122.168} C_VEL
LIN {X 0,Y 597.047,Z 449.404,A -85,B 0,C 180,E1 19120.552,E2 19120.552} C_VEL
LIN {X 0,Y 593.325,Z 429.837,A -85,B 0,C 180,E1 19119.727,E2 19119.727} C_VEL
LIN {X 0,Y 580.928,Z 411.028,A -85,B 0,C 180,E1 19117.726,E2 19117.726} C_VEL
LIN {X 0,Y 568.484,Z 393.248,A -85,B 0,C 180,E1 19115.543,E2 19115.543} C_VEL
LIN {X 0,Y 563.952,Z 386.805,A -85,B 0,C 180,E1 19114.648,E2 19114.648} C_VEL
LIN {X 0,Y 558.16,Z 375.22,A -85,B 0,C 180,E1 19112.387,E2 19112.387} C_VEL
LIN {X 0,Y 553.57,Z 366.468,A -85,B 0,C 180,E1 19110.502,E2 19110.502} C_VEL
LIN {X 0,Y 550.624,Z 361.046,A -85,B 0,C 180,E1 19109.241,E2 19109.241} C_VEL
LIN {X 0,Y 548.523,Z 357.107,A -85,B 0,C 180,E1 19108.291,E2 19108.291} C_VEL
LIN {X 0,Y 546.055,Z 352.478,A -85,B 0,C 180,E1 19107.126,E2 19107.126} C_VEL
LIN {X 0,Y 543.826,Z 348.605,A -85,B 0,C 180,E1 19106.068,E2 19106.068} C_VEL
LIN {X 0,Y 540.82,Z 343.317,A -85,B 0,C 180,E1 19104.548,E2 19104.548} C_VEL
LIN {X 0,Y 537.854,Z 338.413,A -85,B 0,C 180,E1 19102.979,E2 19102.979} C_VEL
LIN {X 0,Y 537.619,Z 337.427,A -85,B 0,C 180,E1 19102.643,E2 19102.643} C_VEL
LIN {X 0,Y 537.616,Z 337.201,A -85,B 0,C 180,E1 19099.333,E2 19099.333} C_VEL
LIN {X 0,Y 537.619,Z 337.257,A -85,B 0,C 180,E1 19095.867,E2 19095.867} C_VEL
LIN {X 0,Y 537.6,Z 337.19,A -85,B 0,C 180,E1 19092.46,E2 19092.46} C_VEL
LIN {X 0,Y 537.616,Z 337.253,A -85,B 0,C 180,E1 19089.044,E2 19089.044} C_VEL
LIN {X 0,Y 537.61,Z 337.194,A -85,B 0,C 180,E1 19085.55,E2 19085.55} C_VEL
LIN {X 0,Y 537.612,Z 337.226,A -85,B 0,C 180,E1 19082.132,E2 19082.132} C_VEL
LIN {X 0,Y 537.604,Z 337.209,A -85,B 0,C 180,E1 19078.721,E2 19078.721} C_VEL
LIN {X 0,Y 537.601,Z 337.211,A -85,B 0,C 180,E1 19075.306,E2 19075.306} C_VEL
LIN {X 0,Y 537.622,Z 337.223,A -85,B 0,C 180,E1 19071.982,E2 19071.982} C_VEL
LIN {X 0,Y 537.586,Z 337.199,A -85,B 0,C 180,E1 19068.629,E2 19068.629} C_VEL
LIN {X 0,Y 537.596,Z 337.263,A -85,B 0,C 180,E1 19065.127,E2 19065.127} C_VEL
LIN {X 0,Y 537.62,Z 337.193,A -85,B 0,C 180,E1 19061.793,E2 19061.793} C_VEL
LIN {X 0,Y 537.607,Z 337.436,A -85,B 0,C 180,E1 19058.906,E2 19058.906} C_VEL
LIN {X 0,Y 539.063,Z 340.897,A -85,B 0,C 180,E1 19057.88,E2 19057.88} C_VEL
LIN {X 0,Y 540.73,Z 342.903,A -85,B 0,C 180,E1 19057.15,E2 19057.15} C_VEL
LIN {X 0,Y 542.446,Z 346.508,A -85,B 0,C 180,E1 19056.191,E2 19056.191} C_VEL
LIN {X 0,Y 543.905,Z 348.486,A -85,B 0,C 180,E1 19055.567,E2 19055.567} C_VEL
LIN {X 0,Y 545.814,Z 352.197,A -85,B 0,C 180,E1 19054.617,E2 19054.617} C_VEL
LIN {X 0,Y 547.029,Z 354.09,A -85,B 0,C 180,E1 19054.096,E2 19054.096} C_VEL
LIN {X 0,Y 550.074,Z 359.681,A -85,B 0,C 180,E1 19052.737,E2 19052.737} C_VEL
LIN {X 0,Y 555.44,Z 366.322,A -85,B 0,C 180,E1 19051.566,E2 19051.566} C_VEL
LIN {X 0,Y 563.134,Z 375.744,A -85,B 0,C 180,E1 19050.041,E2 19050.041} C_VEL
LIN {X 0,Y 571.371,Z 386.27,A -85,B 0,C 180,E1 19048.508,E2 19048.508} C_VEL
LIN {X 0,Y 582.717,Z 401.32,A -85,B 0,C 180,E1 19046.548,E2 19046.548} C_VEL
LIN {X 0,Y 595.188,Z 419.187,A -85,B 0,C 180,E1 19044.549,E2 19044.549} C_VEL
LIN {X 0,Y 601.684,Z 429.076,A -85,B 0,C 180,E1 19043.563,E2 19043.563} C_VEL
LIN {X 0,Y 594.404,Z 633.653,A -85,B 0,C 180,E1 19040.54,E2 19040.54} C_VEL
LIN {X 0,Y 587.802,Z 826.582,A -85,B 0,C 180,E1 19037.723,E2 19037.723} C_VEL
LIN {X 0,Y 586.064,Z 853.569,A -85,B 0,C 180,E1 19037.215,E2 19037.215} C_VEL
LIN {X 0,Y 583.661,Z 880.228,A -85,B 0,C 180,E1 19036.524,E2 19036.524} C_VEL
LIN {X 0,Y 581.353,Z 902.191,A -85,B 0,C 180,E1 19035.824,E2 19035.824} C_VEL
LIN {X 0,Y 578.852,Z 923.49,A -85,B 0,C 180,E1 19035.019,E2 19035.019} C_VEL
LIN {X 0,Y 575.487,Z 949.5,A -85,B 0,C 180,E1 19033.858,E2 19033.858} C_VEL
LIN {X 0,Y 571.909,Z 973.523,A -85,B 0,C 180,E1 19032.578,E2 19032.578} C_VEL
LIN {X 0,Y 568.783,Z 993.306,A -85,B 0,C 180,E1 19031.374,E2 19031.374} C_VEL
LIN {X 0,Y 565.972,Z 1010.151,A -85,B 0,C 180,E1 19030.225,E2 19030.225} C_VEL
LIN {X 0,Y 562.974,Z 1027.237,A -85,B 0,C 180,E1 19028.929,E2 19028.929} C_VEL
LIN {X 0,Y 559.72,Z 1045.34,A -85,B 0,C 180,E1 19027.399,E2 19027.399} C_VEL
LIN {X 0,Y 555.766,Z 1066.967,A -85,B 0,C 180,E1 19025.338,E2 19025.338} C_VEL
LIN {X 0,Y 552.455,Z 1083.995,A -85,B 0,C 180,E1 19023.45,E2 19023.45} C_VEL
LIN {X 0,Y 549.389,Z 1099.665,A -85,B 0,C 180,E1 19021.489,E2 19021.489} C_VEL
LIN {X 0,Y 546.81,Z 1113.37,A -85,B 0,C 180,E1 19019.585,E2 19019.585} C_VEL
LIN {X 0,Y 544.262,Z 1127.871,A -85,B 0,C 180,E1 19017.34,E2 19017.34} C_VEL
LIN {X 0,Y 541.641,Z 1143.693,A -85,B 0,C 180,E1 19014.541,E2 19014.541} C_VEL
LIN {X 0,Y 539.931,Z 1155.292,A -85,B 0,C 180,E1 19012.188,E2 19012.188} C_VEL
LIN {X 0,Y 538.612,Z 1165.438,A -85,B 0,C 180,E1 19009.86,E2 19009.86} C_VEL
LIN {X 0,Y 537.473,Z 1175.941,A -85,B 0,C 180,E1 19007.093,E2 19007.093} C_VEL
LIN {X 0,Y 536.703,Z 1184.855,A -85,B 0,C 180,E1 19004.236,E2 19004.236} C_VEL
LIN {X 0,Y 536.298,Z 1191.132,A -85,B 0,C 180,E1 19001.81,E2 19001.81} C_VEL
LIN {X 0,Y 536.067,Z 1196.322,A -85,B 0,C 180,E1 18999.339,E2 18999.339} C_VEL
LIN {X 0,Y 535.953,Z 1200.783,A -85,B 0,C 180,E1 18996.534,E2 18996.534} C_VEL
LIN {X 0,Y 535.913,Z 1203.565,A -85,B 0,C 180,E1 18993.744,E2 18993.744} C_VEL
LIN {X 0,Y 535.915,Z 1204.736,A -85,B 0,C 180,E1 18991.283,E2 18991.283} C_VEL
LIN {X 0,Y 535.908,Z 1204.803,A -85,B 0,C 180,E1 18989.038,E2 18989.038} C_VEL
LIN {X 0,Y 535.917,Z 1203.904,A -85,B 0,C 180,E1 18986.791,E2 18986.791} C_VEL
LIN {X 0,Y 535.932,Z 1201.866,A -85,B 0,C 180,E1 18984.432,E2 18984.432} C_VEL
LIN {X 0,Y 536.011,Z 1198.247,A -85,B 0,C 180,E1 18981.741,E2 18981.741} C_VEL
LIN {X 0,Y 536.216,Z 1192.484,A -85,B 0,C 180,E1 18978.768,E2 18978.768} C_VEL
LIN {X 0,Y 536.619,Z 1186.065,A -85,B 0,C 180,E1 18976.202,E2 18976.202} C_VEL
LIN {X 0,Y 537.165,Z 1178.972,A -85,B 0,C 180,E1 18973.842,E2 18973.842} C_VEL
LIN {X 0,Y 538.065,Z 1170.27,A -85,B 0,C 180,E1 18971.36,E2 18971.36} C_VEL
LIN {X 0,Y 539.596,Z 1157.834,A -85,B 0,C 180,E1 18968.361,E2 18968.361} C_VEL
LIN {X 0,Y 541.19,Z 1146.563,A -85,B 0,C 180,E1 18966.017,E2 18966.017} C_VEL
LIN {X 0,Y 543.016,Z 1135.085,A -85,B 0,C 180,E1 18963.891,E2 18963.891} C_VEL
LIN {X 0,Y 545.339,Z 1121.564,A -85,B 0,C 180,E1 18961.649,E2 18961.649} C_VEL
LIN {X 0,Y 548.772,Z 1103.042,A -85,B 0,C 180,E1 18958.96,E2 18958.96} C_VEL
LIN {X 0,Y 551.786,Z 1087.284,A -85,B 0,C 180,E1 18956.945,E2 18956.945} C_VEL
LIN {X 0,Y 554.649,Z 1072.744,A -85,B 0,C 180,E1 18955.273,E2 18955.273} C_VEL
LIN {X 0,Y 557.707,Z 1056.158,A -85,B 0,C 180,E1 18953.599,E2 18953.599} C_VEL
LIN {X 0,Y 561.681,Z 1034.743,A -85,B 0,C 180,E1 18951.673,E2 18951.673} C_VEL
LIN {X 0,Y 565.564,Z 1012.506,A -85,B 0,C 180,E1 18949.944,E2 18949.944} C_VEL
LIN {X 0,Y 568.603,Z 994.38,A -85,B 0,C 180,E1 18948.695,E2 18948.695} C_VEL
LIN {X 0,Y 571.607,Z 975.406,A -85,B 0,C 180,E1 18947.53,E2 18947.53} C_VEL
LIN {X 0,Y 574.581,Z 955.367,A -85,B 0,C 180,E1 18946.44,E2 18946.44} C_VEL
LIN {X 0,Y 578.15,Z 929.523,A -85,B 0,C 180,E1 18945.226,E2 18945.226} C_VEL
LIN {X 0,Y 581.107,Z 904.5,A -85,B 0,C 180,E1 18944.257,E2 18944.257} C_VEL
LIN {X 0,Y 583.455,Z 882.231,A -85,B 0,C 180,E1 18943.535,E2 18943.535} C_VEL
LIN {X 0,Y 585.502,Z 859.749,A -85,B 0,C 180,E1 18942.933,E2 18942.933} C_VEL
LIN {X 0,Y 587.578,Z 831.214,A -85,B 0,C 180,E1 18942.351,E2 18942.351} C_VEL
LIN {X 0,Y 589.491,Z 779.675,A -85,B 0,C 180,E1 18941.584,E2 18941.584} C_VEL
LIN {X 0,Y 597.214,Z 553.494,A -85,B 0,C 180,E1 18938.282,E2 18938.282} C_VEL
LIN {X 0,Y 601.619,Z 428.778,A -85,B 0,C 180,E1 18936.427,E2 18936.427} C_VEL
LIN {X 0,Y 588.599,Z 409.613,A -85,B 0,C 180,E1 18934.421,E2 18934.421} C_VEL
LIN {X 0,Y 577.125,Z 393.817,A -85,B 0,C 180,E1 18932.515,E2 18932.515} C_VEL
LIN {X 0,Y 565.56,Z 378.721,A -85,B 0,C 180,E1 18930.433,E2 18930.433} C_VEL
LIN {X 0,Y 556.047,Z 367.079,A -85,B 0,C 180,E1 18928.576,E2 18928.576} C_VEL
LIN {X 0,Y 551.475,Z 361.599,A -85,B 0,C 180,E1 18927.627,E2 18927.627} C_VEL
LIN {X 0,Y 549.805,Z 359.105,A -85,B 0,C 180,E1 18927.16,E2 18927.16} C_VEL
LIN {X 0,Y 546.298,Z 352.759,A -85,B 0,C 180,E1 18925.592,E2 18925.592} C_VEL
LIN {X 0,Y 544.017,Z 348.863,A -85,B 0,C 180,E1 18924.544,E2 18924.544} C_VEL
LIN {X 0,Y 543.15,Z 347.319,A -85,B 0,C 180,E1 18924.122,E2 18924.122} C_VEL
LIN {X 0,Y 541.141,Z 344.152,A -85,B 0,C 180,E1 18923.177,E2 18923.177} C_VEL
LIN {X 0,Y 540.193,Z 342.203,A -85,B 0,C 180,E1 18922.644,E2 18922.644} C_VEL
LIN {X 0,Y 537.879,Z 338.645,A -85,B 0,C 180,E1 18921.482,E2 18921.482} C_VEL
LIN {X 0,Y 537.602,Z 337.398,A -85,B 0,C 180,E1 18921.037,E2 18921.037} C_VEL
LIN {X 0,Y 537.585,Z 337.198,A -85,B 0,C 180,E1 18917.648,E2 18917.648} C_VEL
LIN {X 0,Y 537.629,Z 337.236,A -85,B 0,C 180,E1 18914.314,E2 18914.314} C_VEL
LIN {X 0,Y 537.586,Z 337.208,A -85,B 0,C 180,E1 18910.936,E2 18910.936} C_VEL
LIN {X 0,Y 537.607,Z 337.21,A -85,B 0,C 180,E1 18907.559,E2 18907.559} C_VEL
LIN {X 0,Y 537.618,Z 337.226,A -85,B 0,C 180,E1 18904.16,E2 18904.16} C_VEL
LIN {X 0,Y 537.592,Z 337.201,A -85,B 0,C 180,E1 18900.853,E2 18900.853} C_VEL
LIN {X 0,Y 537.617,Z 337.242,A -85,B 0,C 180,E1 18897.442,E2 18897.442} C_VEL
LIN {X 0,Y 537.61,Z 337.187,A -85,B 0,C 180,E1 18894.022,E2 18894.022} C_VEL
LIN {X 0,Y 537.613,Z 337.259,A -85,B 0,C 180,E1 18890.58,E2 18890.58} C_VEL
LIN {X 0,Y 537.614,Z 337.188,A -85,B 0,C 180,E1 18887.104,E2 18887.104} C_VEL
LIN {X 0,Y 537.608,Z 337.245,A -85,B 0,C 180,E1 18883.8,E2 18883.8} C_VEL
LIN {X 0,Y 537.615,Z 337.207,A -85,B 0,C 180,E1 18880.328,E2 18880.328} C_VEL
LIN {X 0,Y 537.636,Z 337.461,A -85,B 0,C 180,E1 18877.184,E2 18877.184} C_VEL
LIN {X 0,Y 539.289,Z 341.188,A -85,B 0,C 180,E1 18876.043,E2 18876.043} C_VEL
LIN {X 0,Y 540.849,Z 343.396,A -85,B 0,C 180,E1 18875.303,E2 18875.303} C_VEL
LIN {X 0,Y 542.929,Z 347.132,A -85,B 0,C 180,E1 18874.232,E2 18874.232} C_VEL
LIN {X 0,Y 543.844,Z 348.667,A -85,B 0,C 180,E1 18873.794,E2 18873.794} C_VEL
LIN {X 0,Y 546.048,Z 352.467,A -85,B 0,C 180,E1 18872.756,E2 18872.756} C_VEL
LIN {X 0,Y 549.085,Z 357.785,A -85,B 0,C 180,E1 18871.385,E2 18871.385} C_VEL
LIN {X 0,Y 554.836,Z 368.871,A -85,B 0,C 180,E1 18868.854,E2 18868.854} C_VEL
LIN {X 0,Y 559.579,Z 378.062,A -85,B 0,C 180,E1 18866.933,E2 18866.933} C_VEL
LIN {X 0,Y 564.587,Z 387.89,A -85,B 0,C 180,E1 18865.08,E2 18865.08} C_VEL
LIN {X 0,Y 575.713,Z 403.434,A -85,B 0,C 180,E1 18863.063,E2 18863.063} C_VEL
LIN {X 0,Y 588.281,Z 422.065,A -85,B 0,C 180,E1 18860.969,E2 18860.969} C_VEL
LIN {X 0,Y 593.553,Z 430.506,A -85,B 0,C 180,E1 18860.134,E2 18860.134} C_VEL
LIN {X 0,Y 597.091,Z 450.72,A -85,B 0,C 180,E1 18859.321,E2 18859.321} C_VEL
LIN {X 0,Y 589.61,Z 684.454,A -85,B 0,C 180,E1 18856.029,E2 18856.029} C_VEL
LIN {X 0,Y 586.604,Z 786.106,A -85,B 0,C 180,E1 18854.622,E2 18854.622} C_VEL
LIN {X 0,Y 585.735,Z 793.812,A -85,B 0,C 180,E1 18854.586,E2 18854.586} C_VEL
LIN {X 0,Y 580.869,Z 814.427,A -85,B 0,C 180,E1 18854.755,E2 18854.755} C_VEL
LIN {X 0,Y 580.063,Z 821.027,A -85,B 0,C 180,E1 18854.712,E2 18854.712} C_VEL
LIN {X 0,Y 578.734,Z 845.479,A -85,B 0,C 180,E1 18854.301,E2 18854.301} C_VEL
LIN {X 0,Y 577.04,Z 866.421,A -85,B 0,C 180,E1 18853.838,E2 18853.838} C_VEL
LIN {X 0,Y 574.564,Z 891.664,A -85,B 0,C 180,E1 18853.116,E2 18853.116} C_VEL
LIN {X 0,Y 571.575,Z 915.352,A -85,B 0,C 180,E1 18852.248,E2 18852.248} C_VEL
LIN {X 0,Y 568.724,Z 935.247,A -85,B 0,C 180,E1 18851.38,E2 18851.38} C_VEL
LIN {X 0,Y 565.319,Z 956.87,A -85,B 0,C 180,E1 18850.275,E2 18850.275} C_VEL
LIN {X 0,Y 561.179,Z 980.475,A -85,B 0,C 180,E1 18848.842,E2 18848.842} C_VEL
LIN {X 0,Y 557.711,Z 998.744,A -85,B 0,C 180,E1 18847.558,E2 18847.558} C_VEL
LIN {X 0,Y 554.215,Z 1016.389,A -85,B 0,C 180,E1 18846.154,E2 18846.154} C_VEL
LIN {X 0,Y 550.044,Z 1036.81,A -85,B 0,C 180,E1 18844.3,E2 18844.3} C_VEL
LIN {X 0,Y 546.244,Z 1054.543,A -85,B 0,C 180,E1 18842.434,E2 18842.434} C_VEL
LIN {X 0,Y 543.067,Z 1069.406,A -85,B 0,C 180,E1 18840.664,E2 18840.664} C_VEL
LIN {X 0,Y 539.653,Z 1086.008,A -85,B 0,C 180,E1 18838.436,E2 18838.436} C_VEL
LIN {X 0,Y 536.585,Z 1101.183,A -85,B 0,C 180,E1 18836.08,E2 18836.08} C_VEL
LIN {X 0,Y 534.266,Z 1113.964,A -85,B 0,C 180,E1 18833.844,E2 18833.844} C_VEL
LIN {X 0,Y 532.063,Z 1127.427,A -85,B 0,C 180,E1 18831.15,E2 18831.15} C_VEL
LIN {X 0,Y 530.561,Z 1137.972,A -85,B 0,C 180,E1 18828.686,E2 18828.686} C_VEL
LIN {X 0,Y 529.53,Z 1146.704,A -85,B 0,C 180,E1 18826.341,E2 18826.341} C_VEL
LIN {X 0,Y 528.673,Z 1156.092,A -85,B 0,C 180,E1 18823.341,E2 18823.341} C_VEL
LIN {X 0,Y 528.256,Z 1162.291,A -85,B 0,C 180,E1 18820.911,E2 18820.911} C_VEL
LIN {X 0,Y 528.053,Z 1167.07,A -85,B 0,C 180,E1 18818.603,E2 18818.603} C_VEL
LIN {X 0,Y 527.928,Z 1171.329,A -85,B 0,C 180,E1 18815.87,E2 18815.87} C_VEL
LIN {X 0,Y 527.905,Z 1173.768,A -85,B 0,C 180,E1 18813.258,E2 18813.258} C_VEL
LIN {X 0,Y 527.907,Z 1174.789,A -85,B 0,C 180,E1 18810.977,E2 18810.977} C_VEL
LIN {X 0,Y 527.911,Z 1174.743,A -85,B 0,C 180,E1 18808.698,E2 18808.698} C_VEL
LIN {X 0,Y 527.909,Z 1173.421,A -85,B 0,C 180,E1 18806.09,E2 18806.09} C_VEL
LIN {X 0,Y 527.957,Z 1170.371,A -85,B 0,C 180,E1 18803.366,E2 18803.366} C_VEL
LIN {X 0,Y 528.061,Z 1166.62,A -85,B 0,C 180,E1 18801.068,E2 18801.068} C_VEL
LIN {X 0,Y 528.28,Z 1161.735,A -85,B 0,C 180,E1 18798.759,E2 18798.759} C_VEL
LIN {X 0,Y 528.816,Z 1154.263,A -85,B 0,C 180,E1 18795.928,E2 18795.928} C_VEL
LIN {X 0,Y 529.624,Z 1145.835,A -85,B 0,C 180,E1 18793.324,E2 18793.324} C_VEL
LIN {X 0,Y 530.633,Z 1137.371,A -85,B 0,C 180,E1 18791.074,E2 18791.074} C_VEL
LIN {X 0,Y 532.322,Z 1125.772,A -85,B 0,C 180,E1 18788.399,E2 18788.399} C_VEL
LIN {X 0,Y 534.384,Z 1113.202,A -85,B 0,C 180,E1 18785.928,E2 18785.928} C_VEL
LIN {X 0,Y 536.625,Z 1100.972,A -85,B 0,C 180,E1 18783.795,E2 18783.795} C_VEL
LIN {X 0,Y 539.845,Z 1085.002,A -85,B 0,C 180,E1 18781.334,E2 18781.334} C_VEL
LIN {X 0,Y 543.117,Z 1069.176,A -85,B 0,C 180,E1 18779.217,E2 18779.217} C_VEL
LIN {X 0,Y 546.2,Z 1054.74,A -85,B 0,C 180,E1 18777.498,E2 18777.498} C_VEL
LIN {X 0,Y 550.115,Z 1036.516,A -85,B 0,C 180,E1 18775.58,E2 18775.58} C_VEL
LIN {X 0,Y 554.293,Z 1016.029,A -85,B 0,C 180,E1 18773.725,E2 18773.725} C_VEL
LIN {X 0,Y 557.662,Z 999.056,A -85,B 0,C 180,E1 18772.374,E2 18772.374} C_VEL
LIN {X 0,Y 561.127,Z 980.805,A -85,B 0,C 180,E1 18771.089,E2 18771.089} C_VEL
LIN {X 0,Y 565.268,Z 957.257,A -85,B 0,C 180,E1 18769.654,E2 18769.654} C_VEL
LIN {X 0,Y 568.677,Z 935.675,A -85,B 0,C 180,E1 18768.549,E2 18768.549} C_VEL
LIN {X 0,Y 571.488,Z 916.116,A -85,B 0,C 180,E1 18767.692,E2 18767.692} C_VEL
LIN {X 0,Y 574.145,Z 895.159,A -85,B 0,C 180,E1 18766.914,E2 18766.914} C_VEL
LIN {X 0,Y 576.871,Z 868.787,A -85,B 0,C 180,E1 18766.131,E2 18766.131} C_VEL
LIN {X 0,Y 578.629,Z 847.237,A -85,B 0,C 180,E1 18765.642,E2 18765.642} C_VEL
LIN {X 0,Y 579.871,Z 825.578,A -85,B 0,C 180,E1 18765.266,E2 18765.266} C_VEL
LIN {X 0,Y 587.342,Z 590.591,A -85,B 0,C 180,E1 18761.971,E2 18761.971} C_VEL
LIN {X 0,Y 592.024,Z 451.463,A -85,B 0,C 180,E1 18759.973,E2 18759.973} C_VEL
LIN {X 0,Y 588.861,Z 434.658,A -85,B 0,C 180,E1 18759.251,E2 18759.251} C_VEL
LIN {X 0,Y 575.559,Z 414.396,A -85,B 0,C 180,E1 18757.042,E2 18757.042} C_VEL
LIN {X 0,Y 564.406,Z 398.589,A -85,B 0,C 180,E1 18755.029,E2 18755.029} C_VEL
LIN {X 0,Y 555.668,Z 386.338,A -85,B 0,C 180,E1 18753.287,E2 18753.287} C_VEL
LIN {X 0,Y 548.907,Z 373.089,A -85,B 0,C 180,E1 18750.503,E2 18750.503} C_VEL
LIN {X 0,Y 543.714,Z 363.447,A -85,B 0,C 180,E1 18748.205,E2 18748.205} C_VEL
LIN {X 0,Y 540.995,Z 358.509,A -85,B 0,C 180,E1 18746.925,E2 18746.925} C_VEL
LIN {X 0,Y 538.853,Z 354.52,A -85,B 0,C 180,E1 18745.849,E2 18745.849} C_VEL
LIN {X 0,Y 536.101,Z 349.832,A -85,B 0,C 180,E1 18744.46,E2 18744.46} C_VEL
LIN {X 0,Y 534.594,Z 347.577,A -85,B 0,C 180,E1 18743.712,E2 18743.712} C_VEL
LIN {X 0,Y 532.405,Z 343.379,A -85,B 0,C 180,E1 18742.411,E2 18742.411} C_VEL
LIN {X 0,Y 530.077,Z 339.911,A -85,B 0,C 180,E1 18741.118,E2 18741.118} C_VEL
LIN {X 0,Y 529.68,Z 338.392,A -85,B 0,C 180,E1 18740.556,E2 18740.556} C_VEL
LIN {X 0,Y 529.678,Z 338.193,A -85,B 0,C 180,E1 18737.22,E2 18737.22} C_VEL
LIN {X 0,Y 529.674,Z 338.193,A -85,B 0,C 180,E1 18733.871,E2 18733.871} C_VEL
LIN {X 0,Y 529.67,Z 338.223,A -85,B 0,C 180,E1 18730.331,E2 18730.331} C_VEL
LIN {X 0,Y 529.669,Z 338.175,A -85,B 0,C 180,E1 18726.939,E2 18726.939} C_VEL
LIN {X 0,Y 529.676,Z 338.25,A -85,B 0,C 180,E1 18723.463,E2 18723.463} C_VEL
LIN {X 0,Y 529.669,Z 338.174,A -85,B 0,C 180,E1 18720,E2 18720} C_VEL
LIN {X 0,Y 529.674,Z 338.244,A -85,B 0,C 180,E1 18716.537,E2 18716.537} C_VEL
LIN {X 0,Y 529.649,Z 338.184,A -85,B 0,C 180,E1 18713.06,E2 18713.06} C_VEL
LIN {X 0,Y 529.679,Z 338.209,A -85,B 0,C 180,E1 18709.669,E2 18709.669} C_VEL
LIN {X 0,Y 529.668,Z 338.202,A -85,B 0,C 180,E1 18706.24,E2 18706.24} C_VEL
LIN {X 0,Y 529.638,Z 338.191,A -85,B 0,C 180,E1 18702.872,E2 18702.872} C_VEL
LIN {X 0,Y 529.681,Z 338.481,A -85,B 0,C 180,E1 18700.939,E2 18700.939} C_VEL
LIN {X 0,Y 531.267,Z 342.099,A -85,B 0,C 180,E1 18699.738,E2 18699.738} C_VEL
LIN {X 0,Y 532.969,Z 344.312,A -85,B 0,C 180,E1 18698.887,E2 18698.887} C_VEL
LIN {X 0,Y 534.842,Z 347.84,A -85,B 0,C 180,E1 18697.812,E2 18697.812} C_VEL
LIN {X 0,Y 536.158,Z 349.768,A -85,B 0,C 180,E1 18697.176,E2 18697.176} C_VEL
LIN {X 0,Y 538.232,Z 353.475,A -85,B 0,C 180,E1 18696.11,E2 18696.11} C_VEL
LIN {X 0,Y 539.143,Z 354.903,A -85,B 0,C 180,E1 18695.687,E2 18695.687} C_VEL
LIN {X 0,Y 541.334,Z 358.871,A -85,B 0,C 180,E1 18694.626,E2 18694.626} C_VEL
LIN {X 0,Y 542.878,Z 361.481,A -85,B 0,C 180,E1 18694.03,E2 18694.03} C_VEL
LIN {X 0,Y 548.266,Z 367.89,A -85,B 0,C 180,E1 18692.816,E2 18692.816} C_VEL
LIN {X 0,Y 556.261,Z 377.513,A -85,B 0,C 180,E1 18691.142,E2 18691.142} C_VEL
LIN {X 0,Y 567.593,Z 391.943,A -85,B 0,C 180,E1 18688.954,E2 18688.954} C_VEL
LIN {X 0,Y 580.426,Z 409.289,A -85,B 0,C 180,E1 18686.694,E2 18686.694} C_VEL
LIN {X 0,Y 593.368,Z 428.02,A -85,B 0,C 180,E1 18684.602,E2 18684.602} C_VEL
LIN {X 0,Y 596.553,Z 433.058,A -85,B 0,C 180,E1 18684.107,E2 18684.107} C_VEL
LIN {X 0,Y 588.857,Z 640.213,A -85,B 0,C 180,E1 18681.027,E2 18681.027} C_VEL
LIN {X 0,Y 582.162,Z 826.421,A -85,B 0,C 180,E1 18678.284,E2 18678.284} C_VEL
LIN {X 0,Y 580.355,Z 853.322,A -85,B 0,C 180,E1 18677.775,E2 18677.775} C_VEL
LIN {X 0,Y 577.847,Z 879.935,A -85,B 0,C 180,E1 18677.081,E2 18677.081} C_VEL
LIN {X 0,Y 575.437,Z 901.626,A -85,B 0,C 180,E1 18676.383,E2 18676.383} C_VEL
LIN {X 0,Y 572.8,Z 922.804,A -85,B 0,C 180,E1 18675.573,E2 18675.573} C_VEL
LIN {X 0,Y 569.323,Z 948.624,A -85,B 0,C 180,E1 18674.416,E2 18674.416} C_VEL
LIN {X 0,Y 565.501,Z 973.313,A -85,B 0,C 180,E1 18673.093,E2 18673.093} C_VEL
LIN {X 0,Y 562.428,Z 992.051,A -85,B 0,C 180,E1 18671.947,E2 18671.947} C_VEL
LIN {X 0,Y 559.294,Z 1010.13,A -85,B 0,C 180,E1 18670.71,E2 18670.71} C_VEL
LIN {X 0,Y 556.104,Z 1027.802,A -85,B 0,C 180,E1 18669.362,E2 18669.362} C_VEL
LIN {X 0,Y 552.394,Z 1047.676,A -85,B 0,C 180,E1 18667.654,E2 18667.654} C_VEL
LIN {X 0,Y 548.182,Z 1069.405,A -85,B 0,C 180,E1 18665.516,E2 18665.516} C_VEL
LIN {X 0,Y 544.983,Z 1085.882,A -85,B 0,C 180,E1 18663.682,E2 18663.682} C_VEL
LIN {X 0,Y 542.607,Z 1097.973,A -85,B 0,C 180,E1 18662.178,E2 18662.178} C_VEL
LIN {X 0,Y 539.819,Z 1111.826,A -85,B 0,C 180,E1 18660.252,E2 18660.252} C_VEL
LIN {X 0,Y 537.292,Z 1125.067,A -85,B 0,C 180,E1 18658.208,E2 18658.208} C_VEL
LIN {X 0,Y 534.856,Z 1138.892,A -85,B 0,C 180,E1 18655.822,E2 18655.822} C_VEL
LIN {X 0,Y 532.455,Z 1153.711,A -85,B 0,C 180,E1 18652.874,E2 18652.874} C_VEL
LIN {X 0,Y 530.994,Z 1164.06,A -85,B 0,C 180,E1 18650.502,E2 18650.502} C_VEL
LIN {X 0,Y 529.89,Z 1173.105,A -85,B 0,C 180,E1 18648.14,E2 18648.14} C_VEL
LIN {X 0,Y 529.005,Z 1182.071,A -85,B 0,C 180,E1 18645.426,E2 18645.426} C_VEL
LIN {X 0,Y 528.384,Z 1190.059,A -85,B 0,C 180,E1 18642.456,E2 18642.456} C_VEL
LIN {X 0,Y 528.114,Z 1195.492,A -85,B 0,C 180,E1 18639.921,E2 18639.921} C_VEL
LIN {X 0,Y 527.983,Z 1199.523,A -85,B 0,C 180,E1 18637.508,E2 18637.508} C_VEL
LIN {X 0,Y 527.926,Z 1202.581,A -85,B 0,C 180,E1 18634.965,E2 18634.965} C_VEL
LIN {X 0,Y 527.911,Z 1204.577,A -85,B 0,C 180,E1 18632.062,E2 18632.062} C_VEL
LIN {X 0,Y 527.896,Z 1204.871,A -85,B 0,C 180,E1 18629.349,E2 18629.349} C_VEL
LIN {X 0,Y 527.916,Z 1204.037,A -85,B 0,C 180,E1 18626.96,E2 18626.96} C_VEL
LIN {X 0,Y 527.931,Z 1202.091,A -85,B 0,C 180,E1 18624.566,E2 18624.566} C_VEL
LIN {X 0,Y 527.995,Z 1199.043,A -85,B 0,C 180,E1 18622.163,E2 18622.163} C_VEL
LIN {X 0,Y 528.172,Z 1194.252,A -85,B 0,C 180,E1 18619.419,E2 18619.419} C_VEL
LIN {X 0,Y 528.59,Z 1187.274,A -85,B 0,C 180,E1 18616.434,E2 18616.434} C_VEL
LIN {X 0,Y 529.145,Z 1180.208,A -85,B 0,C 180,E1 18613.985,E2 18613.985} C_VEL
LIN {X 0,Y 529.992,Z 1172.23,A -85,B 0,C 180,E1 18611.617,E2 18611.617} C_VEL
LIN {X 0,Y 531.114,Z 1163.144,A -85,B 0,C 180,E1 18609.272,E2 18609.272} C_VEL
LIN {X 0,Y 532.956,Z 1150.574,A -85,B 0,C 180,E1 18606.446,E2 18606.446} C_VEL
LIN {X 0,Y 535.175,Z 1136.988,A -85,B 0,C 180,E1 18603.837,E2 18603.837} C_VEL
LIN {X 0,Y 537.465,Z 1124.122,A -85,B 0,C 180,E1 18601.638,E2 18601.638} C_VEL
LIN {X 0,Y 540.144,Z 1110.281,A -85,B 0,C 180,E1 18599.522,E2 18599.522} C_VEL
LIN {X 0,Y 543.858,Z 1091.896,A -85,B 0,C 180,E1 18597.03,E2 18597.03} C_VEL
LIN {X 0,Y 547.254,Z 1074.142,A -85,B 0,C 180,E1 18594.991,E2 18594.991} C_VEL
LIN {X 0,Y 550.417,Z 1057.697,A -85,B 0,C 180,E1 18593.298,E2 18593.298} C_VEL
LIN {X 0,Y 553.784,Z 1040.078,A -85,B 0,C 180,E1 18591.669,E2 18591.669} C_VEL
LIN {X 0,Y 557.847,Z 1018.425,A -85,B 0,C 180,E1 18589.892,E2 18589.892} C_VEL
LIN {X 0,Y 561.845,Z 995.443,A -85,B 0,C 180,E1 18588.273,E2 18588.273} C_VEL
LIN {X 0,Y 565.069,Z 975.928,A -85,B 0,C 180,E1 18587.058,E2 18587.058} C_VEL
LIN {X 0,Y 568.152,Z 955.983,A -85,B 0,C 180,E1 18585.961,E2 18585.961} C_VEL
LIN {X 0,Y 571.771,Z 930.974,A -85,B 0,C 180,E1 18584.766,E2 18584.766} C_VEL
LIN {X 0,Y 575.038,Z 905.101,A -85,B 0,C 180,E1 18583.741,E2 18583.741} C_VEL
LIN {X 0,Y 577.49,Z 883.257,A -85,B 0,C 180,E1 18583.018,E2 18583.018} C_VEL
LIN {X 0,Y 579.556,Z 861.841,A -85,B 0,C 180,E1 18582.432,E2 18582.432} C_VEL
LIN {X 0,Y 581.461,Z 838.08,A -85,B 0,C 180,E1 18581.918,E2 18581.918} C_VEL
LIN {X 0,Y 583.185,Z 801.757,A -85,B 0,C 180,E1 18581.34,E2 18581.34} C_VEL
LIN {X 0,Y 591.216,Z 575.524,A -85,B 0,C 180,E1 18578.018,E2 18578.018} C_VEL
LIN {X 0,Y 596.465,Z 432.757,A -85,B 0,C 180,E1 18575.881,E2 18575.881} C_VEL
LIN {X 0,Y 584.082,Z 414.526,A -85,B 0,C 180,E1 18573.923,E2 18573.923} C_VEL
LIN {X 0,Y 573.257,Z 399.558,A -85,B 0,C 180,E1 18572.081,E2 18572.081} C_VEL
LIN {X 0,Y 562.549,Z 385.451,A -85,B 0,C 180,E1 18570.111,E2 18570.111} C_VEL
LIN {X 0,Y 552.586,Z 373.095,A -85,B 0,C 180,E1 18568.123,E2 18568.123} C_VEL
LIN {X 0,Y 544.97,Z 364.001,A -85,B 0,C 180,E1 18566.478,E2 18566.478} C_VEL
LIN {X 0,Y 542.241,Z 360.432,A -85,B 0,C 180,E1 18565.797,E2 18565.797} C_VEL
LIN {X 0,Y 539.093,Z 354.788,A -85,B 0,C 180,E1 18564.315,E2 18564.315} C_VEL
LIN {X 0,Y 536.218,Z 349.955,A -85,B 0,C 180,E1 18562.904,E2 18562.904} C_VEL
LIN {X 0,Y 535.242,Z 348.304,A -85,B 0,C 180,E1 18562.402,E2 18562.402} C_VEL
LIN {X 0,Y 533.203,Z 345.002,A -85,B 0,C 180,E1 18561.334,E2 18561.334} C_VEL
LIN {X 0,Y 532.288,Z 343.285,A -85,B 0,C 180,E1 18560.796,E2 18560.796} C_VEL
LIN {X 0,Y 529.978,Z 339.725,A -85,B 0,C 180,E1 18559.508,E2 18559.508} C_VEL
LIN {X 0,Y 529.669,Z 338.419,A -85,B 0,C 180,E1 18559.062,E2 18559.062} C_VEL
LIN {X 0,Y 529.681,Z 338.216,A -85,B 0,C 180,E1 18555.998,E2 18555.998} C_VEL
LIN {X 0,Y 529.66,Z 338.18,A -85,B 0,C 180,E1 18552.649,E2 18552.649} C_VEL
LIN {X 0,Y 529.653,Z 338.254,A -85,B 0,C 180,E1 18549.234,E2 18549.234} C_VEL
LIN {X 0,Y 529.676,Z 338.174,A -85,B 0,C 180,E1 18545.851,E2 18545.851} C_VEL
LIN {X 0,Y 529.677,Z 338.239,A -85,B 0,C 180,E1 18542.38,E2 18542.38} C_VEL
LIN {X 0,Y 529.654,Z 338.183,A -85,B 0,C 180,E1 18538.918,E2 18538.918} C_VEL
LIN {X 0,Y 529.677,Z 338.213,A -85,B 0,C 180,E1 18535.561,E2 18535.561} C_VEL
LIN {X 0,Y 529.676,Z 338.19,A -85,B 0,C 180,E1 18532.079,E2 18532.079} C_VEL
LIN {X 0,Y 529.667,Z 338.19,A -85,B 0,C 180,E1 18528.678,E2 18528.678} C_VEL
LIN {X 0,Y 529.679,Z 338.221,A -85,B 0,C 180,E1 18525.236,E2 18525.236} C_VEL
LIN {X 0,Y 529.661,Z 338.181,A -85,B 0,C 180,E1 18521.723,E2 18521.723} C_VEL
LIN {X 0,Y 529.702,Z 338.47,A -85,B 0,C 180,E1 18519.214,E2 18519.214} C_VEL
LIN {X 0,Y 531.25,Z 342.072,A -85,B 0,C 180,E1 18518.004,E2 18518.004} C_VEL
LIN {X 0,Y 532.95,Z 344.27,A -85,B 0,C 180,E1 18517.147,E2 18517.147} C_VEL
LIN {X 0,Y 535.024,Z 348.11,A -85,B 0,C 180,E1 18515.957,E2 18515.957} C_VEL
LIN {X 0,Y 536.085,Z 349.78,A -85,B 0,C 180,E1 18515.422,E2 18515.422} C_VEL
LIN {X 0,Y 538.407,Z 353.765,A -85,B 0,C 180,E1 18514.242,E2 18514.242} C_VEL
LIN {X 0,Y 541.257,Z 358.812,A -85,B 0,C 180,E1 18512.852,E2 18512.852} C_VEL
LIN {X 0,Y 544.843,Z 365.678,A -85,B 0,C 180,E1 18511.141,E2 18511.141} C_VEL
LIN {X 0,Y 547.47,Z 370.684,A -85,B 0,C 180,E1 18509.962,E2 18509.962} C_VEL
LIN {X 0,Y 551.759,Z 378.653,A -85,B 0,C 180,E1 18508.174,E2 18508.174} C_VEL
LIN {X 0,Y 556.184,Z 387.193,A -85,B 0,C 180,E1 18506.47,E2 18506.47} C_VEL
LIN {X 0,Y 568.831,Z 404.766,A -85,B 0,C 180,E1 18504.048,E2 18504.048} C_VEL
LIN {X 0,Y 581.166,Z 422.842,A -85,B 0,C 180,E1 18501.902,E2 18501.902} C_VEL
LIN {X 0,Y 589.109,Z 435.438,A -85,B 0,C 180,E1 18500.603,E2 18500.603} C_VEL
LIN {X 0,Y 592.055,Z 452.71,A -85,B 0,C 180,E1 18499.902,E2 18499.902} C_VEL
LIN {X 0,Y 584.248,Z 685.834,A -85,B 0,C 180,E1 18496.597,E2 18496.597} C_VEL
LIN {X 0,Y 580.063,Z 821.027,A -85,B 0,C 180,E1 18494.712,E2 18494.712} C_VEL
LIN {X 0,Y 578.997,Z 828.707,A -85,B 0,C 180,E1 18494.671,E2 18494.671} C_VEL
LIN {X 0,Y 573.769,Z 848.112,A -85,B 0,C 180,E1 18494.767,E2 18494.767} C_VEL
LIN {X 0,Y 572.503,Z 855.718,A -85,B 0,C 180,E1 18494.679,E2 18494.679} C_VEL
LIN {X 0,Y 570.031,Z 881.036,A -85,B 0,C 180,E1 18494.019,E2 18494.019} C_VEL
LIN {X 0,Y 567.756,Z 900.684,A -85,B 0,C 180,E1 18493.38,E2 18493.38} C_VEL
LIN {X 0,Y 565.23,Z 919.578,A -85,B 0,C 180,E1 18492.65,E2 18492.65} C_VEL
LIN {X 0,Y 561.768,Z 942.681,A -85,B 0,C 180,E1 18491.598,E2 18491.598} C_VEL
LIN {X 0,Y 557.76,Z 965.763,A -85,B 0,C 180,E1 18490.327,E2 18490.327} C_VEL
LIN {X 0,Y 554.297,Z 984.26,A -85,B 0,C 180,E1 18489.15,E2 18489.15} C_VEL
LIN {X 0,Y 550.675,Z 1002.541,A -85,B 0,C 180,E1 18487.828,E2 18487.828} C_VEL
LIN {X 0,Y 545.976,Z 1024.954,A -85,B 0,C 180,E1 18485.955,E2 18485.955} C_VEL
LIN {X 0,Y 542.211,Z 1042.174,A -85,B 0,C 180,E1 18484.294,E2 18484.294} C_VEL
LIN {X 0,Y 538.712,Z 1058.07,A -85,B 0,C 180,E1 18482.565,E2 18482.565} C_VEL
LIN {X 0,Y 534.75,Z 1076.176,A -85,B 0,C 180,E1 18480.321,E2 18480.321} C_VEL
LIN {X 0,Y 531.475,Z 1091.107,A -85,B 0,C 180,E1 18478.178,E2 18478.178} C_VEL
LIN {X 0,Y 528.699,Z 1104.429,A -85,B 0,C 180,E1 18476.025,E2 18476.025} C_VEL
LIN {X 0,Y 525.893,Z 1119.191,A -85,B 0,C 180,E1 18473.295,E2 18473.295} C_VEL
LIN {X 0,Y 523.993,Z 1130.362,A -85,B 0,C 180,E1 18470.906,E2 18470.906} C_VEL
LIN {X 0,Y 522.564,Z 1140.142,A -85,B 0,C 180,E1 18468.52,E2 18468.52} C_VEL
LIN {X 0,Y 521.287,Z 1150.744,A -85,B 0,C 180,E1 18465.463,E2 18465.463} C_VEL
LIN {X 0,Y 520.62,Z 1157.838,A -85,B 0,C 180,E1 18462.986,E2 18462.986} C_VEL
LIN {X 0,Y 520.222,Z 1163.676,A -85,B 0,C 180,E1 18460.521,E2 18460.521} C_VEL
LIN {X 0,Y 520.005,Z 1168.815,A -85,B 0,C 180,E1 18457.736,E2 18457.736} C_VEL
LIN {X 0,Y 519.923,Z 1172.126,A -85,B 0,C 180,E1 18455.186,E2 18455.186} C_VEL
LIN {X 0,Y 519.905,Z 1173.972,A -85,B 0,C 180,E1 18452.977,E2 18452.977} C_VEL
LIN {X 0,Y 519.899,Z 1174.834,A -85,B 0,C 180,E1 18450.772,E2 18450.772} C_VEL
LIN {X 0,Y 519.907,Z 1174.652,A -85,B 0,C 180,E1 18448.237,E2 18448.237} C_VEL
LIN {X 0,Y 519.905,Z 1172.79,A -85,B 0,C 180,E1 18445.367,E2 18445.367} C_VEL
LIN {X 0,Y 519.958,Z 1170.051,A -85,B 0,C 180,E1 18443.042,E2 18443.042} C_VEL
LIN {X 0,Y 520.114,Z 1166.085,A -85,B 0,C 180,E1 18440.596,E2 18440.596} C_VEL
LIN {X 0,Y 520.502,Z 1159.544,A -85,B 0,C 180,E1 18437.576,E2 18437.576} C_VEL
LIN {X 0,Y 521.105,Z 1152.384,A -85,B 0,C 180,E1 18434.988,E2 18434.988} C_VEL
LIN {X 0,Y 521.92,Z 1145.011,A -85,B 0,C 180,E1 18432.726,E2 18432.726} C_VEL
LIN {X 0,Y 523.349,Z 1134.709,A -85,B 0,C 180,E1 18430.002,E2 18430.002} C_VEL
LIN {X 0,Y 525.222,Z 1122.918,A -85,B 0,C 180,E1 18427.384,E2 18427.384} C_VEL
LIN {X 0,Y 527.351,Z 1111.285,A -85,B 0,C 180,E1 18425.108,E2 18425.108} C_VEL
LIN {X 0,Y 530.446,Z 1096.077,A -85,B 0,C 180,E1 18422.496,E2 18422.496} C_VEL
LIN {X 0,Y 533.519,Z 1081.647,A -85,B 0,C 180,E1 18420.346,E2 18420.346} C_VEL
LIN {X 0,Y 536.713,Z 1067.148,A -85,B 0,C 180,E1 18418.433,E2 18418.433} C_VEL
LIN {X 0,Y 540.82,Z 1048.821,A -85,B 0,C 180,E1 18416.303,E2 18416.303} C_VEL
LIN {X 0,Y 544.853,Z 1030.076,A -85,B 0,C 180,E1 18414.428,E2 18414.428} C_VEL
LIN {X 0,Y 548.553,Z 1012.685,A -85,B 0,C 180,E1 18412.891,E2 18412.891} C_VEL
LIN {X 0,Y 552.894,Z 991.72,A -85,B 0,C 180,E1 18411.265,E2 18411.265} C_VEL
LIN {X 0,Y 557.052,Z 969.638,A -85,B 0,C 180,E1 18409.814,E2 18409.814} C_VEL
LIN {X 0,Y 560.314,Z 951.032,A -85,B 0,C 180,E1 18408.748,E2 18408.748} C_VEL
LIN {X 0,Y 563.738,Z 929.839,A -85,B 0,C 180,E1 18407.7,E2 18407.7} C_VEL
LIN {X 0,Y 567.334,Z 904.143,A -85,B 0,C 180,E1 18406.65,E2 18406.65} C_VEL
LIN {X 0,Y 569.841,Z 882.854,A -85,B 0,C 180,E1 18405.942,E2 18405.942} C_VEL
LIN {X 0,Y 572.045,Z 860.522,A -85,B 0,C 180,E1 18405.342,E2 18405.342} C_VEL
LIN {X 0,Y 574.089,Z 832.342,A -85,B 0,C 180,E1 18404.787,E2 18404.787} C_VEL
LIN {X 0,Y 576.857,Z 751.921,A -85,B 0,C 180,E1 18403.641,E2 18403.641} C_VEL
LIN {X 0,Y 584.397,Z 528.514,A -85,B 0,C 180,E1 18400.476,E2 18400.476} C_VEL
LIN {X 0,Y 587.017,Z 453.316,A -85,B 0,C 180,E1 18399.375,E2 18399.375} C_VEL
LIN {X 0,Y 584.552,Z 439.822,A -85,B 0,C 180,E1 18398.791,E2 18398.791} C_VEL
LIN {X 0,Y 572.237,Z 420.807,A -85,B 0,C 180,E1 18396.698,E2 18396.698} C_VEL
LIN {X 0,Y 561.207,Z 405.01,A -85,B 0,C 180,E1 18394.667,E2 18394.667} C_VEL
LIN {X 0,Y 551.436,Z 391.589,A -85,B 0,C 180,E1 18392.708,E2 18392.708} C_VEL
LIN {X 0,Y 546.83,Z 385.085,A -85,B 0,C 180,E1 18391.654,E2 18391.654} C_VEL
LIN {X 0,Y 542.827,Z 377.484,A -85,B 0,C 180,E1 18389.946,E2 18389.946} C_VEL
LIN {X 0,Y 538.911,Z 369.791,A -85,B 0,C 180,E1 18388.117,E2 18388.117} C_VEL
LIN {X 0,Y 535.95,Z 364.528,A -85,B 0,C 180,E1 18386.719,E2 18386.719} C_VEL
LIN {X 0,Y 533.165,Z 359.527,A -85,B 0,C 180,E1 18385.315,E2 18385.315} C_VEL
LIN {X 0,Y 530.56,Z 354.781,A -85,B 0,C 180,E1 18383.903,E2 18383.903} C_VEL
LIN {X 0,Y 528.408,Z 351.114,A -85,B 0,C 180,E1 18382.707,E2 18382.707} C_VEL
LIN {X 0,Y 527.242,Z 349.273,A -85,B 0,C 180,E1 18382.055,E2 18382.055} C_VEL
LIN {X 0,Y 525.153,Z 345.522,A -85,B 0,C 180,E1 18380.741,E2 18380.741} C_VEL
LIN {X 0,Y 523.463,Z 343.236,A -85,B 0,C 180,E1 18379.761,E2 18379.761} C_VEL
LIN {X 0,Y 521.755,Z 339.431,A -85,B 0,C 180,E1 18378.26,E2 18378.26} C_VEL
LIN {X 0,Y 521.749,Z 339.221,A -85,B 0,C 180,E1 18375.015,E2 18375.015} C_VEL
LIN {X 0,Y 521.732,Z 339.172,A -85,B 0,C 180,E1 18371.497,E2 18371.497} C_VEL
LIN {X 0,Y 521.729,Z 339.188,A -85,B 0,C 180,E1 18368.153,E2 18368.153} C_VEL
LIN {X 0,Y 521.734,Z 339.187,A -85,B 0,C 180,E1 18364.727,E2 18364.727} C_VEL
LIN {X 0,Y 521.724,Z 339.174,A -85,B 0,C 180,E1 18361.318,E2 18361.318} C_VEL
LIN {X 0,Y 521.739,Z 339.209,A -85,B 0,C 180,E1 18357.913,E2 18357.913} C_VEL
LIN {X 0,Y 521.728,Z 339.165,A -85,B 0,C 180,E1 18354.501,E2 18354.501} C_VEL
LIN {X 0,Y 521.719,Z 339.238,A -85,B 0,C 180,E1 18351.069,E2 18351.069} C_VEL
LIN {X 0,Y 521.737,Z 339.162,A -85,B 0,C 180,E1 18347.605,E2 18347.605} C_VEL
LIN {X 0,Y 521.732,Z 339.21,A -85,B 0,C 180,E1 18344.166,E2 18344.166} C_VEL
LIN {X 0,Y 521.796,Z 339.704,A -85,B 0,C 180,E1 18343.181,E2 18343.181} C_VEL
LIN {X 0,Y 523.453,Z 343.202,A -85,B 0,C 180,E1 18341.859,E2 18341.859} C_VEL
LIN {X 0,Y 525.158,Z 345.484,A -85,B 0,C 180,E1 18340.884,E2 18340.884} C_VEL
LIN {X 0,Y 527.259,Z 349.268,A -85,B 0,C 180,E1 18339.578,E2 18339.578} C_VEL
LIN {X 0,Y 528.307,Z 350.677,A -85,B 0,C 180,E1 18339.04,E2 18339.04} C_VEL
LIN {X 0,Y 530.386,Z 354.489,A -85,B 0,C 180,E1 18337.849,E2 18337.849} C_VEL
LIN {X 0,Y 531.446,Z 356.147,A -85,B 0,C 180,E1 18337.313,E2 18337.313} C_VEL
LIN {X 0,Y 533.763,Z 360.129,A -85,B 0,C 180,E1 18336.132,E2 18336.132} C_VEL
LIN {X 0,Y 535.239,Z 362.671,A -85,B 0,C 180,E1 18335.557,E2 18335.557} C_VEL
LIN {X 0,Y 540.098,Z 368.194,A -85,B 0,C 180,E1 18334.387,E2 18334.387} C_VEL
LIN {X 0,Y 548.908,Z 378.766,A -85,B 0,C 180,E1 18332.41,E2 18332.41} C_VEL
LIN {X 0,Y 560.907,Z 393.802,A -85,B 0,C 180,E1 18329.968,E2 18329.968} C_VEL
LIN {X 0,Y 572.531,Z 409.51,A -85,B 0,C 180,E1 18327.814,E2 18327.814} C_VEL
LIN {X 0,Y 584.252,Z 426.029,A -85,B 0,C 180,E1 18325.822,E2 18325.822} C_VEL
LIN {X 0,Y 591.472,Z 437.157,A -85,B 0,C 180,E1 18324.658,E2 18324.658} C_VEL
LIN {X 0,Y 583.406,Z 645.321,A -85,B 0,C 180,E1 18321.544,E2 18321.544} C_VEL
LIN {X 0,Y 576.595,Z 826.37,A -85,B 0,C 180,E1 18318.856,E2 18318.856} C_VEL
LIN {X 0,Y 574.721,Z 853.213,A -85,B 0,C 180,E1 18318.346,E2 18318.346} C_VEL
LIN {X 0,Y 572.12,Z 879.765,A -85,B 0,C 180,E1 18317.65,E2 18317.65} C_VEL
LIN {X 0,Y 569.669,Z 900.951,A -85,B 0,C 180,E1 18316.966,E2 18316.966} C_VEL
LIN {X 0,Y 566.953,Z 921.872,A -85,B 0,C 180,E1 18316.162,E2 18316.162} C_VEL
LIN {X 0,Y 563.822,Z 943.737,A -85,B 0,C 180,E1 18315.182,E2 18315.182} C_VEL
LIN {X 0,Y 559.53,Z 970.803,A -85,B 0,C 180,E1 18313.754,E2 18313.754} C_VEL
LIN {X 0,Y 556.121,Z 990.797,A -85,B 0,C 180,E1 18312.534,E2 18312.534} C_VEL
LIN {X 0,Y 552.888,Z 1008.717,A -85,B 0,C 180,E1 18311.306,E2 18311.306} C_VEL
LIN {X 0,Y 549.58,Z 1026.357,A -85,B 0,C 180,E1 18309.958,E2 18309.958} C_VEL
LIN {X 0,Y 546.002,Z 1044.905,A -85,B 0,C 180,E1 18308.374,E2 18308.374} C_VEL
LIN {X 0,Y 541.952,Z 1065.535,A -85,B 0,C 180,E1 18306.381,E2 18306.381} C_VEL
LIN {X 0,Y 538.07,Z 1084.528,A -85,B 0,C 180,E1 18304.267,E2 18304.267} C_VEL
LIN {X 0,Y 535.091,Z 1099.323,A -85,B 0,C 180,E1 18302.431,E2 18302.431} C_VEL
LIN {X 0,Y 532.758,Z 1111.054,A -85,B 0,C 180,E1 18300.821,E2 18300.821} C_VEL
LIN {X 0,Y 530.043,Z 1124.364,A -85,B 0,C 180,E1 18298.753,E2 18298.753} C_VEL
LIN {X 0,Y 527.757,Z 1136.35,A -85,B 0,C 180,E1 18296.68,E2 18296.68} C_VEL
LIN {X 0,Y 525.48,Z 1149.422,A -85,B 0,C 180,E1 18294.148,E2 18294.148} C_VEL
LIN {X 0,Y 523.401,Z 1162.681,A -85,B 0,C 180,E1 18291.165,E2 18291.165} C_VEL
LIN {X 0,Y 522.187,Z 1171.889,A -85,B 0,C 180,E1 18288.765,E2 18288.765} C_VEL
LIN {X 0,Y 521.283,Z 1179.858,A -85,B 0,C 180,E1 18286.377,E2 18286.377} C_VEL
LIN {X 0,Y 520.665,Z 1186.97,A -85,B 0,C 180,E1 18283.889,E2 18283.889} C_VEL
LIN {X 0,Y 520.194,Z 1194.112,A -85,B 0,C 180,E1 18280.819,E2 18280.819} C_VEL
LIN {X 0,Y 520.005,Z 1198.982,A -85,B 0,C 180,E1 18277.999,E2 18277.999} C_VEL
LIN {X 0,Y 519.934,Z 1202.089,A -85,B 0,C 180,E1 18275.518,E2 18275.518} C_VEL
LIN {X 0,Y 519.916,Z 1204.035,A -85,B 0,C 180,E1 18273.087,E2 18273.087} C_VEL
LIN {X 0,Y 519.895,Z 1204.894,A -85,B 0,C 180,E1 18270.551,E2 18270.551} C_VEL
LIN {X 0,Y 519.908,Z 1204.438,A -85,B 0,C 180,E1 18267.575,E2 18267.575} C_VEL
LIN {X 0,Y 519.929,Z 1202.429,A -85,B 0,C 180,E1 18264.814,E2 18264.814} C_VEL
LIN {X 0,Y 519.985,Z 1199.519,A -85,B 0,C 180,E1 18262.375,E2 18262.375} C_VEL
LIN {X 0,Y 520.129,Z 1195.488,A -85,B 0,C 180,E1 18259.925,E2 18259.925} C_VEL
LIN {X 0,Y 520.426,Z 1190.052,A -85,B 0,C 180,E1 18257.348,E2 18257.348} C_VEL
LIN {X 0,Y 521.089,Z 1181.973,A -85,B 0,C 180,E1 18254.303,E2 18254.303} C_VEL
LIN {X 0,Y 522.042,Z 1173.102,A -85,B 0,C 180,E1 18251.577,E2 18251.577} C_VEL
LIN {X 0,Y 523.153,Z 1164.519,A -85,B 0,C 180,E1 18249.293,E2 18249.293} C_VEL
LIN {X 0,Y 524.687,Z 1154.228,A -85,B 0,C 180,E1 18246.885,E2 18246.885} C_VEL
LIN {X 0,Y 527.109,Z 1140.162,A -85,B 0,C 180,E1 18244.012,E2 18244.012} C_VEL
LIN {X 0,Y 529.767,Z 1125.763,A -85,B 0,C 180,E1 18241.477,E2 18241.477} C_VEL
LIN {X 0,Y 532.423,Z 1112.591,A -85,B 0,C 180,E1 18239.407,E2 18239.407} C_VEL
LIN {X 0,Y 534.731,Z 1101.074,A -85,B 0,C 180,E1 18237.797,E2 18237.797} C_VEL
LIN {X 0,Y 537.767,Z 1085.976,A -85,B 0,C 180,E1 18235.904,E2 18235.904} C_VEL
LIN {X 0,Y 541.163,Z 1069.22,A -85,B 0,C 180,E1 18234.016,E2 18234.016} C_VEL
LIN {X 0,Y 545.654,Z 1046.814,A -85,B 0,C 180,E1 18231.797,E2 18231.797} C_VEL
LIN {X 0,Y 549.396,Z 1027.365,A -85,B 0,C 180,E1 18230.123,E2 18230.123} C_VEL
LIN {X 0,Y 552.889,Z 1008.714,A -85,B 0,C 180,E1 18228.693,E2 18228.693} C_VEL
LIN {X 0,Y 556.419,Z 989.092,A -85,B 0,C 180,E1 18227.354,E2 18227.354} C_VEL
LIN {X 0,Y 560.796,Z 962.943,A -85,B 0,C 180,E1 18225.802,E2 18225.802} C_VEL
LIN {X 0,Y 564.317,Z 940.242,A -85,B 0,C 180,E1 18224.651,E2 18224.651} C_VEL
LIN {X 0,Y 567.225,Z 919.885,A -85,B 0,C 180,E1 18223.756,E2 18223.756} C_VEL
LIN {X 0,Y 569.972,Z 898.516,A -85,B 0,C 180,E1 18222.949,E2 18222.949} C_VEL
LIN {X 0,Y 573.036,Z 871.224,A -85,B 0,C 180,E1 18222.104,E2 18222.104} C_VEL
LIN {X 0,Y 575.239,Z 845.969,A -85,B 0,C 180,E1 18221.505,E2 18221.505} C_VEL
LIN {X 0,Y 576.732,Z 823.617,A -85,B 0,C 180,E1 18221.1,E2 18221.1} C_VEL
LIN {X 0,Y 584.876,Z 606.112,A -85,B 0,C 180,E1 18217.873,E2 18217.873} C_VEL
LIN {X 0,Y 591.372,Z 436.83,A -85,B 0,C 180,E1 18215.328,E2 18215.328} C_VEL
LIN {X 0,Y 578.983,Z 418.503,A -85,B 0,C 180,E1 18213.311,E2 18213.311} C_VEL
LIN {X 0,Y 567.124,Z 402.189,A -85,B 0,C 180,E1 18211.222,E2 18211.222} C_VEL
LIN {X 0,Y 558.388,Z 390.765,A -85,B 0,C 180,E1 18209.56,E2 18209.56} C_VEL
LIN {X 0,Y 549.596,Z 379.681,A -85,B 0,C 180,E1 18207.759,E2 18207.759} C_VEL
LIN {X 0,Y 542.392,Z 371.015,A -85,B 0,C 180,E1 18206.171,E2 18206.171} C_VEL
LIN {X 0,Y 538.166,Z 365.943,A -85,B 0,C 180,E1 18205.181,E2 18205.181} C_VEL
LIN {X 0,Y 534.478,Z 361.47,A -85,B 0,C 180,E1 18204.245,E2 18204.245} C_VEL
LIN {X 0,Y 533.185,Z 359.444,A -85,B 0,C 180,E1 18203.661,E2 18203.661} C_VEL
LIN {X 0,Y 530.647,Z 354.794,A -85,B 0,C 180,E1 18202.305,E2 18202.305} C_VEL
LIN {X 0,Y 528.39,Z 350.949,A -85,B 0,C 180,E1 18201.072,E2 18201.072} C_VEL
LIN {X 0,Y 525.214,Z 345.669,A -85,B 0,C 180,E1 18199.22,E2 18199.22} C_VEL
LIN {X 0,Y 524.154,Z 344.006,A -85,B 0,C 180,E1 18198.577,E2 18198.577} C_VEL
LIN {X 0,Y 521.982,Z 340.518,A -85,B 0,C 180,E1 18197.157,E2 18197.157} C_VEL
LIN {X 0,Y 521.751,Z 339.363,A -85,B 0,C 180,E1 18196.625,E2 18196.625} C_VEL
LIN {X 0,Y 521.701,Z 339.177,A -85,B 0,C 180,E1 18193.184,E2 18193.184} C_VEL
LIN {X 0,Y 521.737,Z 339.221,A -85,B 0,C 180,E1 18189.709,E2 18189.709} C_VEL
LIN {X 0,Y 521.739,Z 339.16,A -85,B 0,C 180,E1 18186.271,E2 18186.271} C_VEL
LIN {X 0,Y 521.724,Z 339.242,A -85,B 0,C 180,E1 18182.746,E2 18182.746} C_VEL
LIN {X 0,Y 521.725,Z 339.163,A -85,B 0,C 180,E1 18179.231,E2 18179.231} C_VEL
LIN {X 0,Y 521.737,Z 339.21,A -85,B 0,C 180,E1 18175.824,E2 18175.824} C_VEL
LIN {X 0,Y 521.738,Z 339.171,A -85,B 0,C 180,E1 18172.29,E2 18172.29} C_VEL
LIN {X 0,Y 521.73,Z 339.18,A -85,B 0,C 180,E1 18168.839,E2 18168.839} C_VEL
LIN {X 0,Y 521.733,Z 339.203,A -85,B 0,C 180,E1 18165.346,E2 18165.346} C_VEL
LIN {X 0,Y 521.74,Z 339.291,A -85,B 0,C 180,E1 18161.797,E2 18161.797} C_VEL
LIN {X 0,Y 521.862,Z 339.953,A -85,B 0,C 180,E1 18161.339,E2 18161.339} C_VEL
LIN {X 0,Y 523.795,Z 343.637,A -85,B 0,C 180,E1 18159.903,E2 18159.903} C_VEL
LIN {X 0,Y 525.126,Z 345.419,A -85,B 0,C 180,E1 18159.141,E2 18159.141} C_VEL
LIN {X 0,Y 526.977,Z 348.971,A -85,B 0,C 180,E1 18157.933,E2 18157.933} C_VEL
LIN {X 0,Y 528.24,Z 350.636,A -85,B 0,C 180,E1 18157.285,E2 18157.285} C_VEL
LIN {X 0,Y 530.29,Z 354.467,A -85,B 0,C 180,E1 18156.084,E2 18156.084} C_VEL
LIN {X 0,Y 531.326,Z 356.159,A -85,B 0,C 180,E1 18155.543,E2 18155.543} C_VEL
LIN {X 0,Y 534.209,Z 361.383,A -85,B 0,C 180,E1 18154.025,E2 18154.025} C_VEL
LIN {X 0,Y 537.045,Z 366.548,A -85,B 0,C 180,E1 18152.621,E2 18152.621} C_VEL
LIN {X 0,Y 540.004,Z 372.074,A -85,B 0,C 180,E1 18151.221,E2 18151.221} C_VEL
LIN {X 0,Y 544.585,Z 380.745,A -85,B 0,C 180,E1 18149.185,E2 18149.185} C_VEL
